FUNCTION_BLOCK "FB_Chute2PEC"
{ S7_Optimized_Access := 'TRUE' }
VERSION : 0.1
// ATTRIBUTES
// AUTO_NUMBER = True
// BLOCK_NUMBER = 204
// END_ATTRIBUTES
   VAR_INPUT
      iUDT_ChuteConfiguration { ExternalAccessible := 'False'; ExternalVisible := 'False'; ExternalWritable := 'False'} : "UDT_Chute2PECConfiguration";   // Chute Configuration structure
      iUDT_UpstreamConveyorStatus { ExternalAccessible := 'False'; ExternalVisible := 'False'; ExternalWritable := 'False'} : "UDT_CommonStatus";   // Upstream conveyor status
      ix_PECFull { ExternalAccessible := 'False'; ExternalVisible := 'False'; ExternalWritable := 'False'} : Bool;   // TRUE when Chute Full photoeye is not blocked
      ix_PECHalfFull { ExternalAccessible := 'False'; ExternalVisible := 'False'; ExternalWritable := 'False'} : Bool;   // TRUE when Chute Half Full photoeye is not blocked
      ix_Disabled { ExternalAccessible := 'False'; ExternalVisible := 'False'; ExternalWritable := 'False'} : Bool;   // TRUE when chute is disabled
      ix_HardwareOk { ExternalAccessible := 'False'; ExternalVisible := 'False'; ExternalWritable := 'False'} : Bool;   // TRUE when chute hardware is Ok
      iudi_DelayHardwareOK { ExternalAccessible := 'False'; ExternalVisible := 'False'; ExternalWritable := 'False'} : UDInt;   // Time to delay for hardware ok signal
   END_VAR

   VAR_OUTPUT
      qx_Lamp { ExternalAccessible := 'False'; ExternalVisible := 'False'; ExternalWritable := 'False'} : Bool;   // Output Chute Lamp half full/ full
      qUDT_HMIStatus { ExternalAccessible := 'False'; ExternalVisible := 'False'; ExternalWritable := 'False'} : "UDT_Chute2PECStatus";   // HMI status structure
      qUDT_Status { ExternalAccessible := 'False'; ExternalVisible := 'False'; ExternalWritable := 'False'} : "UDT_CommonStatus";   // Common status structure
   END_VAR

   VAR_IN_OUT
      iqUDT_EquipmentControl : "UDT_EquipmentControl";   // Equipment control structure
      iqUDT_UpstreamConveyorHandshake : "UDT_ConveyorHandshake";   // Upstream handshake structure
      iqUDT_Statistics : "UDT_Chute2PECStatistics";   // Statistics structure
   END_VAR

   VAR
      sUDT_HMIStatus { ExternalAccessible := 'False'; ExternalVisible := 'False'; ExternalWritable := 'False'; S7_SetPoint := 'False'} : "UDT_Chute2PECStatus";   // HMI status structure
      sUDT_CommonStatus { ExternalAccessible := 'False'; ExternalVisible := 'False'; ExternalWritable := 'False'; S7_SetPoint := 'False'} : "UDT_CommonStatus";   // Common status structure
      sUDT_CommonStatusOld { ExternalAccessible := 'False'; ExternalVisible := 'False'; ExternalWritable := 'False'; S7_SetPoint := 'False'} : "UDT_CommonStatus";   // Auxiliary status structure
      sFB_HardwareOk { ExternalAccessible := 'False'; ExternalVisible := 'False'; ExternalWritable := 'False'; S7_SetPoint := 'False'} : "FB_TimerOnOffDelay";   // Timer on/off delay for hardware ok signal
      sFB_ChuteHalfFullDetectionDelay { ExternalAccessible := 'False'; ExternalVisible := 'False'; ExternalWritable := 'False'; S7_SetPoint := 'False'} : "FB_TimerOnOffDelay";   // Timer on/off delay for chute half  full detection
      sFB_ChuteFullDetectionDelay { ExternalAccessible := 'False'; ExternalVisible := 'False'; ExternalWritable := 'False'; S7_SetPoint := 'False'} : "FB_TimerOnOffDelay";   // Timer on/off delay for chute full detection
      sR_TRIG_HalfFull {InstructionName := 'R_TRIG'; LibVersion := '1.0'; ExternalAccessible := 'False'; ExternalVisible := 'False'; ExternalWritable := 'False'; S7_SetPoint := 'False'} : R_TRIG;   // Rising edge trigger on chute half full signal
      sR_TRIG_Disabled {InstructionName := 'R_TRIG'; LibVersion := '1.0'; ExternalAccessible := 'False'; ExternalVisible := 'False'; ExternalWritable := 'False'; S7_SetPoint := 'False'} : R_TRIG;   // Rising edge trigger on chute disabled signal
      sR_TRIG_ChuteFull {InstructionName := 'R_TRIG'; LibVersion := '1.0'; ExternalAccessible := 'False'; ExternalVisible := 'False'; ExternalWritable := 'False'; S7_SetPoint := 'False'} : R_TRIG;   // Rising edge trigger on chute full signal
      sF_TRIG_UpdateStatus {InstructionName := 'F_TRIG'; LibVersion := '1.0'; ExternalAccessible := 'False'; ExternalVisible := 'False'; ExternalWritable := 'False'; S7_SetPoint := 'False'} : F_TRIG;   // Falling edge trigger on status change
      sx_Full { ExternalAccessible := 'False'; ExternalVisible := 'False'; ExternalWritable := 'False'} : Bool;   // Full status
      sx_HalfFull { ExternalAccessible := 'False'; ExternalVisible := 'False'; ExternalWritable := 'False'} : Bool;   // Half full status
   END_VAR


BEGIN
	(*
	----------------------------------------------------------------------------------------

	Version history:
	Date        | Version   | Author        | Remark
	----------------------------------------------------------------------------------------
	19/10/2021  | 0.1       | J. Krawczuk   | first release TIA 16.0
	29/10/2021  | 0.1       | M. Piela      | Design change, comments corrections
	14/01/2022  | 0.2       | G. Vlooswijk  | Fixed statistics reset
	30/07/2022  | 0.3       | G. Vlooswijk  | Removed running and energy save status for FedEx Scada
	21/02/2023  | 4.0       | F.Baten       | 4.0 Release TIA 17.5
	 *)

	REGION 1 - Timers

	    // Chute full detection timer
	    #sFB_ChuteFullDetectionDelay(iudi_OnDelayTime := #iUDT_ChuteConfiguration.FullDetectionTime,
	                                 iudi_OffDelayTime := #iUDT_ChuteConfiguration.FullReleaseTime,
	                                 ix_SignalToDelay := NOT #ix_PECFull,
	                                 qx_DelayedSignal => #sx_Full);

	    // Chute half full detection timer
	    #sFB_ChuteHalfFullDetectionDelay(iudi_OnDelayTime := #iUDT_ChuteConfiguration.HalfFullDetectionTime,
	                                     iudi_OffDelayTime := #iUDT_ChuteConfiguration.HalfFullReleaseTime,
	                                     ix_SignalToDelay := NOT #ix_PECHalfFull,
	                                     qx_DelayedSignal => #sx_HalfFull);

	    // Hardware ok signal delay
	    #sFB_HardwareOk(iudi_OnDelayTime := #iudi_DelayHardwareOK,
	                    ix_SignalToDelay := #ix_HardwareOk);


	END_REGION

	REGION 2 - Stop upstream conveyor

	    // Stop upstream conveyor when chute is full or disabled
	    #iqUDT_UpstreamConveyorHandshake.RTR := NOT #sx_Full AND NOT #ix_Disabled AND #sFB_HardwareOk.qx_DelayedSignal;

	END_REGION

	REGION 3 - Update output

	    // Update the outputs
	    #qx_Lamp := #sx_Full OR (#sx_HalfFull AND "DB_Memory".Clock_1Hz);

	END_REGION

	REGION 4 - Status

	    // Update chute full specific status
	    #sUDT_HMIStatus.Specific.ChuteFull := #sx_Full AND #sFB_HardwareOk.qx_DelayedSignal;

	    // Update chute half full specific status
	    #sUDT_HMIStatus.Specific.ChuteHalfFull := #sx_HalfFull AND #sFB_HardwareOk.qx_DelayedSignal;

	    //Update chute disabled specific status
	    #sUDT_HMIStatus.Specific.ChuteDisabled := #ix_Disabled AND #sFB_HardwareOk.qx_DelayedSignal;

	    // Update common safety stop
	    #sUDT_CommonStatus.SafetyStop := #iUDT_UpstreamConveyorStatus.SafetyStop;

	    // Update common automatic on
	    #sUDT_CommonStatus.AutoON := #iUDT_UpstreamConveyorStatus.AutoON;

	    // Update common stopped
	    #sUDT_CommonStatus.Stopped := #iUDT_UpstreamConveyorStatus.Stopped;

	    // Update HMI status number for chute disabled
	    IF #sUDT_HMIStatus.Specific.ChuteDisabled AND NOT #sUDT_CommonStatus.SafetyStop
	    THEN
	        #sUDT_HMIStatus.Status := "DB_HMIStatusConfiguration".DisableByManagement;

	    END_IF;

	    // Update HMI status number for chute half full
	    IF #sUDT_HMIStatus.Specific.ChuteHalfFull AND NOT #sUDT_CommonStatus.SafetyStop
	    THEN
	        #sUDT_HMIStatus.Status := "DB_HMIStatusConfiguration".ChuteHalfFull;

	    END_IF;

	    // Update HMI status number for chute full
	    IF #sUDT_HMIStatus.Specific.ChuteFull AND NOT #sUDT_CommonStatus.SafetyStop
	    THEN
	        #sUDT_HMIStatus.Status := "DB_HMIStatusConfiguration".ChuteFull;

	    END_IF;

	    // Collecting F_TRIG on chute full, chute half full or chute disabled status to update common status
	    #sF_TRIG_UpdateStatus(CLK := #sUDT_HMIStatus.Specific.ChuteFull
	                          OR #sUDT_HMIStatus.Specific.ChuteDisabled
	                          OR #sUDT_HMIStatus.Specific.ChuteHalfFull);

	    // HMI status number calculation
	    IF #sUDT_CommonStatusOld <> #sUDT_CommonStatus OR #sF_TRIG_UpdateStatus.Q
	    THEN

	        // Update auto on status number
	        IF #sUDT_CommonStatus.AutoON
	        THEN
	            #sUDT_HMIStatus.Status := "DB_HMIStatusConfiguration".AutoON;

	        END_IF;

	        IF #sUDT_CommonStatus.Stopped
	        THEN
	            #sUDT_HMIStatus.Status := "DB_HMIStatusConfiguration".Stopped;

	        END_IF;

	        IF #sUDT_CommonStatus.SafetyStop
	        THEN
	            #sUDT_HMIStatus.Status := "DB_HMIStatusConfiguration".SafetyStop;

	        END_IF;

	        // Copy common status structure to the old common status structure
	        #sUDT_CommonStatusOld := #sUDT_CommonStatus;
	        #qUDT_Status := #sUDT_CommonStatus;

	    END_IF;

	    #qUDT_HMIStatus := #sUDT_HMIStatus;

	END_REGION

	REGION 5 - Statistics

	    // Chute full R_TRIG for statistics purpose
	    #sR_TRIG_ChuteFull(CLK := #sUDT_HMIStatus.Specific.ChuteFull);

	    // Chute full statistics
	    IF #sUDT_HMIStatus.Specific.ChuteFull
	        OR #iqUDT_EquipmentControl.Command.ResetData
	    THEN
	        "FC_Statistics"(ix_Reset := #iqUDT_EquipmentControl.Command.ResetData,
	                        ix_Activate := #sUDT_HMIStatus.Specific.ChuteFull,
	                        ix_RTrigActivate := #sR_TRIG_ChuteFull.Q,
	                        iqUDT_Statistics := #iqUDT_Statistics.ChuteFull);

	    END_IF;

	    // Chute disabled R_TRIG for statistics purpose
	    #sR_TRIG_Disabled(CLK := #sUDT_HMIStatus.Specific.ChuteDisabled);

	    // Chute disabled statistics
	    IF #sUDT_HMIStatus.Specific.ChuteDisabled
	        OR #iqUDT_EquipmentControl.Command.ResetData
	    THEN
	        "FC_Statistics"(ix_Reset := #iqUDT_EquipmentControl.Command.ResetData,
	                        ix_Activate := #sUDT_HMIStatus.Specific.ChuteDisabled,
	                        ix_RTrigActivate := #sR_TRIG_Disabled.Q,
	                        iqUDT_Statistics := #iqUDT_Statistics.ChuteDisabled);

	    END_IF;

	    // Chute half full R_TRIG for statistics purpose
	    #sR_TRIG_HalfFull(CLK := #sUDT_HMIStatus.Specific.ChuteHalfFull);

	    // Chute half full statistics
	    IF #sUDT_HMIStatus.Specific.ChuteHalfFull
	        OR #iqUDT_EquipmentControl.Command.ResetData
	    THEN

	        "FC_Statistics"(ix_Reset := #iqUDT_EquipmentControl.Command.ResetData,
	                        ix_Activate := #sUDT_HMIStatus.Specific.ChuteHalfFull,
	                        ix_RTrigActivate := #sR_TRIG_HalfFull.Q,
	                        iqUDT_Statistics := #iqUDT_Statistics.ChuteHalfFull);

	    END_IF;

	END_REGION

	REGION 6 - Equipment Report

	    "FC_EquipmentReport"(iUDT_Status := #sUDT_CommonStatus,
	                         iqUDT_Control := #iqUDT_EquipmentControl);

	END_REGION
END_FUNCTION_BLOCK

FUNCTION_BLOCK "FB_PendantVT100"
{ S7_Optimized_Access := 'TRUE' }
VERSION : 0.1
// ATTRIBUTES
// AUTO_NUMBER = True
// BLOCK_NUMBER = 222
// END_ATTRIBUTES
   VAR_INPUT
      iUDT_Configuration { ExternalAccessible := 'False'; ExternalVisible := 'False'; ExternalWritable := 'False'} : "UDT_PendantVT100Configuration" := ([16#001B, 16#005B, 16#0031, 16#003B, 16#0033, 16#0048, 16#006D, 16#0000], [16#001B, 16#005B, 16#0032, 16#003B, 16#0035, 16#0048, 16#006D, 16#0000], (), (), ());
      iUDT_PendantInputs { ExternalAccessible := 'False'; ExternalVisible := 'False'; ExternalWritable := 'False'} : "UDT_PendantVT100InBytes";   //   Input Bytes 1,2 and 3 of HW Config
      ix_HMIDivertSelectionEnabled { ExternalAccessible := 'False'; ExternalVisible := 'False'; ExternalWritable := 'False'} : Bool;   //   When 'TRUE' The divert selection screen is activated from the HMI
      ix_SimulationModeActive { ExternalAccessible := 'False'; ExternalVisible := 'False'; ExternalWritable := 'False'} : Bool;   //   When 'TRUE' Simulation mode active
      ix_LCDDS1 { ExternalAccessible := 'False'; ExternalVisible := 'False'; ExternalWritable := 'False'} : Bool;   //   When 'TRUE' Display is busy writing a message row 1
      ix_PowerOk { ExternalAccessible := 'False'; ExternalVisible := 'False'; ExternalWritable := 'False'} : Bool;   //   When 'TRUE' 24VDC available
      ix_ServiceMode { ExternalAccessible := 'False'; ExternalVisible := 'False'; ExternalWritable := 'False'} : Bool;   //   When 'TRUE' Service Mode ON
      ix_VFDRunFeedback { ExternalAccessible := 'False'; ExternalVisible := 'False'; ExternalWritable := 'False'} : Bool;   //   When 'TRUE' VFD Run
      ix_SorterSTOActive { ExternalAccessible := 'False'; ExternalVisible := 'False'; ExternalWritable := 'False'} : Bool;   //   VFD STO active feedback
      ix_SorterSS1Active { ExternalAccessible := 'False'; ExternalVisible := 'False'; ExternalWritable := 'False'} : Bool;   //   VFD SS1 active feedback
   END_VAR

   VAR_OUTPUT
      qUDT_Display { ExternalAccessible := 'False'; ExternalVisible := 'False'; ExternalWritable := 'False'} : "UDT_PendantVT100LCDOutBytes";   //   Display bytes
      qUDT_HMIStatus { ExternalAccessible := 'False'; ExternalVisible := 'False'; ExternalWritable := 'False'} : "UDT_PendantVT100Status";   //   Configuation variables for VT100 Radio Pendant
      qUDT_Status { ExternalAccessible := 'False'; ExternalVisible := 'False'; ExternalWritable := 'False'} : "UDT_CommonStatus";   //   Common status structure
   END_VAR

   VAR_IN_OUT
      iqUDT_EquipmentControl : "UDT_EquipmentControl";
      iqUDT_PendantInterface : "UDT_PendantVT100Interface";   //   Interface structure
      iqUDT_Statistics : "UDT_PendantVT100Statistics";   //   Staristic structure
      iq_ConveyorInterface : "UDT_ConveyorInterface";
   END_VAR

   VAR
      sUDT_Display { ExternalAccessible := 'False'; ExternalVisible := 'False'; ExternalWritable := 'False'; S7_SetPoint := 'False'} : "UDT_PendantVT100LCDOutBytes";   //    Array of 8 bytes for the display message
      sUDT_CommonStatus { ExternalAccessible := 'False'; ExternalVisible := 'False'; ExternalWritable := 'False'; S7_SetPoint := 'False'} : "UDT_CommonStatus";   //    Common status structure
      sUDT_CommonStatusOld { ExternalAccessible := 'False'; ExternalVisible := 'False'; ExternalWritable := 'False'; S7_SetPoint := 'False'} : "UDT_CommonStatus";   //    Common status structure
      sUDT_HMIStatus { ExternalAccessible := 'False'; ExternalVisible := 'False'; ExternalWritable := 'False'; S7_SetPoint := 'False'} : "UDT_PendantVT100Status";
      sUDT_PNDevice { ExternalAccessible := 'False'; ExternalVisible := 'False'; ExternalWritable := 'False'; S7_SetPoint := 'False'} : "UDT_PNDevice";   //    PN device info structure
      sFB_TimerOnOffDelayCheckSupply { ExternalAccessible := 'False'; ExternalVisible := 'False'; ExternalWritable := 'False'; S7_SetPoint := 'False'} : "FB_TimerOnOffDelay";
      sF_TRIG_Servicemode {InstructionName := 'F_TRIG'; LibVersion := '1.0'; ExternalAccessible := 'False'; ExternalVisible := 'False'; ExternalWritable := 'False'; S7_SetPoint := 'False'} : F_TRIG;   //   Falling edge trigger service mode
      sF_TRIG_DisplayReady {InstructionName := 'F_TRIG'; LibVersion := '1.0'; ExternalAccessible := 'False'; ExternalVisible := 'False'; ExternalWritable := 'False'; S7_SetPoint := 'False'} : F_TRIG;   //   Falling edge trigger display ready
      sR_TRIG_RunCommand {InstructionName := 'R_TRIG'; LibVersion := '1.0'; ExternalAccessible := 'False'; ExternalVisible := 'False'; ExternalWritable := 'False'; S7_SetPoint := 'False'} : R_TRIG;   //   Rising edge trigger run command
      sR_TRIG_PNReceiverNotOnline {InstructionName := 'R_TRIG'; LibVersion := '1.0'; ExternalAccessible := 'False'; ExternalVisible := 'False'; ExternalWritable := 'False'; S7_SetPoint := 'False'} : R_TRIG;   //   Rising edge trigger PN receiver not online
      sR_TRIG_PNReceiverError {InstructionName := 'R_TRIG'; LibVersion := '1.0'; ExternalAccessible := 'False'; ExternalVisible := 'False'; ExternalWritable := 'False'; S7_SetPoint := 'False'} : R_TRIG;   //   Rising edge trigger PN device error
      sR_TRIG_ControlHealthy {InstructionName := 'R_TRIG'; LibVersion := '1.0'; ExternalAccessible := 'False'; ExternalVisible := 'False'; ExternalWritable := 'False'; S7_SetPoint := 'False'} : R_TRIG;   //   Rising edge trigger control healthy
      sa_Int { ExternalAccessible := 'False'; ExternalVisible := 'False'; ExternalWritable := 'False'} : Struct   //   Integer structure
         Step { ExternalAccessible := 'False'; ExternalVisible := 'False'; ExternalWritable := 'False'; S7_SetPoint := 'True'} : Int;   //    Step of the message sequence
      END_STRUCT;
      sa_Bool { ExternalAccessible := 'False'; ExternalVisible := 'False'; ExternalWritable := 'False'} : Struct   //   Bool structure
         DivertUp { ExternalAccessible := 'False'; ExternalVisible := 'False'; ExternalWritable := 'False'} : Bool;   //    When 'TRUE' Any divert is up
         HardwareAvailable { ExternalAccessible := 'False'; ExternalVisible := 'False'; ExternalWritable := 'False'} : Bool;   //    When 'TRUE' Hardware available and ready to use
         PermissionRequested { ExternalAccessible := 'False'; ExternalVisible := 'False'; ExternalWritable := 'False'} : Bool;   //    When 'TRUE' Permission requested for horn to sound
         PermissionGranted { ExternalAccessible := 'False'; ExternalVisible := 'False'; ExternalWritable := 'False'} : Bool;   //    When 'TRUE' Horn sounded before start of VFD
         PowerOk { ExternalAccessible := 'False'; ExternalVisible := 'False'; ExternalWritable := 'False'} : Bool;   //    When 'TRUE' Power is present at receiver
         PNDeviceHealthy { ExternalAccessible := 'False'; ExternalVisible := 'False'; ExternalWritable := 'False'} : Bool;   //    When 'TRUE' Receiver is healthy
         RadioConnection { ExternalAccessible := 'False'; ExternalVisible := 'False'; ExternalWritable := 'False'} : Bool;   //    When 'TRUE' Initial connection with radio
         RunRequest { ExternalAccessible := 'False'; ExternalVisible := 'False'; ExternalWritable := 'False'} : Bool;   //    When 'TRUE' Request to run
         ServiceModeEngaged { ExternalAccessible := 'False'; ExternalVisible := 'False'; ExternalWritable := 'False'} : Bool;   //    True = Service mode is engaged
      END_STRUCT;
   END_VAR

   VAR_TEMP
      ti_index : Int;   //   temporary integer for loops
   END_VAR

   VAR CONSTANT
      cudi_PowerSupplyDelayTime : UDInt := 7000;   //   Power supply delay time [ms]
   END_VAR


BEGIN

	(*
	----------------------------------------------------------------------------------------

	Version history:
	Date        | Version   | Author        | Remark
	----------------------------------------------------------------------------------------
	14/04/2019  | 1.0       | S. Theocharis | first release TIA15.1
	11/09/2019  | 1.1       | S. Theocharis | update for UPS EMA Baseline
	04/11/2019  | 1.2       | S. Theocharis | Key Switch wired@safety input
	30/01/2020  | 3.0       | S. Theocharis | Different button for fast speed,
	                                        | code to activate diverters
	                                        | Status, statistics and equipement control
	                                        | structures added
	04/03/2020  | 3.1       | M. Piela      | Changed comments and subregions names, added constants to timers
	25/06/2020  | 3.2       | L. Klar       | Horn delay deleted
	07/07/2020  | 3.3       | M. Piela      | Delete unused signal from the interface, change condition to enable step 1
	                                        | in service mode
	07/07/2020  | 3.4       | M. Piela      | Added conditions to set the signaling request signal
	28/07/2020  | 3.5       | S. Theocharis | Changed input name
	11/08/2020  | 3.6       | S. Theocharis | Update the divert functionality
	03/06/2021  | 3.7       | S. Theocharis | Force to slow speed for missing pin at service point
	21/02/2023  | 4.0       | F.Baten       | 4.0 Release TIA 17.5
	*)

	REGION Notes
	(*

	Note1:
	 ib_Buttons.xxxxxx1 is  the signal when the associate button is pressed half way
	 ib_buttons.xxxxxx2 is  the signal when the associate button is pressed full

	 Not Pressed:                 Halfway Pressed                    Full way Pressed
	                             ib_Buttons.xxxxxx1 = TRUE           ib_Buttons.xxxxxx1 = TRUE
	                             ib_Buttons.xxxxxx2 = FALSE          ib_Buttons.xxxxxx2 = TRUE
	     ________
	     |      |                        ________
	     |      |                        |      |                       ________
	     |      |                        |      |                       |      |
	 ____|      |____                 ___|      |____                ___|      |____


	 Note2:
	 The block is designed for the following remote controller:
	 Danfoss TM70/1.13DC  (Ikusi)
	 https://www.danfoss.com/en/products/electronic-controls/dps/plus1-remote-controls/transmitters/legacy-handheld-transmitters/
	  *)
	END_REGION

	REGION 1 -  Get Receiver Profinet number

	    "FC_GetDevicePN"(is_PNDeviceName := #iUDT_Configuration.PNDeviceName,
	                     ix_SimulationModeActive := #ix_SimulationModeActive,
	                     iqUDT_PND := #sUDT_PNDevice);

	END_REGION

	REGION 2 - Reset errors

	    IF #iqUDT_EquipmentControl.Command.Reset                         // Reser errors when Reset from HMI or MCP is given
	    THEN
	        #sUDT_HMIStatus.Specific.PNSlaveNotOnline := FALSE;
	        #sUDT_HMIStatus.Specific.PNSlaveError := FALSE;
	        #sUDT_HMIStatus.Specific.CommunicationError := FALSE;          // Not in use
	    END_IF;

	END_REGION

	REGION 3 - Hardware checks
	    // PN Receiver will only be available after the delay, so the device has time for the initialisation
	    #sFB_TimerOnOffDelayCheckSupply(iudi_OnDelayTime := #cudi_PowerSupplyDelayTime,
	                                    ix_SignalToDelay := #ix_PowerOk,
	                                    ix_Enable := TRUE,
	                                    qx_DelayedSignal => #sa_Bool.PowerOk);

	    // Check if PN receiver device is online
	    IF NOT "DB_ProfinetDiagnostic".ProfinetNetworks[#sUDT_PNDevice.PNNetworknumber].DeviceStatus[#sUDT_PNDevice.PNDeviceNumber].DeviceState.Exist
	        AND NOT #ix_SimulationModeActive
	        AND #sa_Bool.PowerOk
	    THEN
	        #sUDT_HMIStatus.Specific.PNSlaveNotOnline := TRUE;
	    END_IF;

	    // Check if PN Receiver device has an error
	    IF "DB_ProfinetDiagnostic".ProfinetNetworks[#sUDT_PNDevice.PNNetworknumber].DeviceStatus[#sUDT_PNDevice.PNDeviceNumber].DeviceState.Error
	        AND NOT #ix_SimulationModeActive
	        AND #sa_Bool.PowerOk
	    THEN
	        #sUDT_HMIStatus.Specific.PNSlaveError := TRUE;
	    END_IF;

	    // Set bit when PN Receiver device is healthy (online and no error)
	    #sa_Bool.PNDeviceHealthy := NOT #sUDT_HMIStatus.Specific.PNSlaveNotOnline
	    AND NOT #sUDT_HMIStatus.Specific.PNSlaveError
	    AND #sUDT_PNDevice.PNDeviceFound
	    AND #sa_Bool.PowerOk;

	    // Set hardware available bit when all conditions are met
	    #sa_Bool.HardwareAvailable := (#sa_Bool.PowerOk
	    AND #sa_Bool.PNDeviceHealthy)
	    OR #ix_SimulationModeActive;

	END_REGION

	REGION 4 -  Detect service mode selection changes

	    //static memory to engage the service mode. Only when the sorter is standstill
	    IF #sa_Bool.HardwareAvailable AND #ix_ServiceMode AND NOT #ix_VFDRunFeedback
	    THEN
	        #sa_Bool.ServiceModeEngaged := TRUE;
	    END_IF;

	    //disengage service mode when hardware is not available or switch is off
	    IF NOT #sa_Bool.HardwareAvailable OR NOT #ix_ServiceMode
	    THEN
	        #sa_Bool.ServiceModeEngaged := FALSE;
	    END_IF;

	    //service mode to interface
	    #iqUDT_PendantInterface.ServiceModeEngaged := #sa_Bool.ServiceModeEngaged;


	    //Detect falling edge of service mode
	    #sF_TRIG_Servicemode(CLK := #sa_Bool.ServiceModeEngaged);

	END_REGION

	REGION 5 -  Service mode

	    IF #sa_Bool.ServiceModeEngaged
	    THEN

	        REGION 5.1 - Detect Tx connection & LCD readiness to receive message

	            #sR_TRIG_ControlHealthy(CLK := #iUDT_PendantInputs.Stop_NC);//Rising edge of communication

	            //set radio Tx-Rx connection
	            IF #sR_TRIG_ControlHealthy.Q
	            THEN    (* or replace it directly with the input #iudt_PendantInputs.Stop_NO) *)
	                #sa_Bool.RadioConnection := True;
	            END_IF;

	            #sF_TRIG_DisplayReady(CLK := #ix_LCDDS1);//LCD Status Signal. When ix_LCD_DS1 is False, the LCD is ready to receive a new message

	        END_REGION

	        REGION 5.2 - LCD messages
	            //First communication established. Activate message one to move cursor in the begin of line 1

	            IF #sa_Bool.RadioConnection
	            THEN
	                #sa_Int.Step := 1;           // step 1 - new message is activated
	                #sa_Bool.RadioConnection := FALSE;
	            END_IF;

	            //reset variables for display. that can be used to move the step to eg 98 and there reset the variables and move the step to 0 again
	            IF NOT #iUDT_PendantInputs.Stop_NC
	            THEN
	                // #st_Int.Step := 98;
	                FOR #ti_index := 0 TO 7 BY 1 DO
	                    #qUDT_Display."Byte"[#ti_index] := b#16#0;
	                    #sUDT_Display."Byte"[#ti_index] := b#16#0;
	                END_FOR;
	            END_IF;

	            // Screen  Messages
	            CASE #sa_Int.Step OF

	                1: // Move Cursor in the Start Point
	                    #sUDT_Display."Byte" := #iUDT_Configuration.Line1Cursor;  // message
	                    #sa_Int.Step := 2;                                 //  is written static memory

	                2: // when display is not busy write the output
	                    IF NOT #ix_LCDDS1
	                    THEN
	                        #qUDT_Display."Byte" := #sUDT_Display."Byte";
	                        #sa_Int.Step := 3;    // move to next step
	                    END_IF;

	                3: //Write PLC name
	                    FOR #ti_index := 0 TO 7 BY 1 DO
	                        #sUDT_Display."Byte"[#ti_index] := CHAR_TO_BYTE(#iUDT_Configuration.DisplayName[#ti_index + 1]);
	                    END_FOR;
	                    #sa_Int.Step := 4;     //move to next step

	                4: //when display is not busy write the output
	                    IF #sF_TRIG_DisplayReady.Q
	                    THEN   (* may need to be replaced with :NOT #ix_LCD_DS1 *)
	                        #qUDT_Display."Byte" := #sUDT_Display."Byte";
	                        #sa_Int.Step := 99;// move to next step
	                    END_IF;
	            END_CASE;

	        END_REGION

	        REGION 5.3 - Output to the sorter control function
	            //Stop Button
	            #iqUDT_PendantInterface.PendantStopHealthy := #iUDT_PendantInputs.Stop_NC AND NOT #iUDT_PendantInputs.Stop_NO;

	            // Reset - Control On
	            #iqUDT_PendantInterface.PendantReset := #iUDT_PendantInputs.ResetButton1;

	        END_REGION

	        REGION 5.4 - Motion control
	            // STO request to safety program
	            #iqUDT_PendantInterface.RequestSTO := #iUDT_PendantInputs.PB_Speed1 OR #iUDT_PendantInputs.PB_Speed2;

	            //Run reuqest condition
	            #sa_Bool.RunRequest := (#iUDT_PendantInputs.PB_Speed2 XOR #iUDT_PendantInputs.PB_Speed1) AND NOT #sa_Bool.DivertUp;

	            //Check permission to run after horn sounded
	            IF #iUDT_Configuration.HornRequest
	            THEN

	                //Detect new run request
	                #sR_TRIG_RunCommand(CLK := #sa_Bool.RunRequest AND NOT #ix_VFDRunFeedback);

	                //On the positie edge of the new run command which requires permission set the control request and reset the permissiong granted bit
	                IF #sR_TRIG_RunCommand.Q AND NOT #ix_SorterSS1Active AND NOT #iq_ConveyorInterface.InternalErrorVFD
	                THEN
	                    #iqUDT_EquipmentControl.Request.SignalingRequest := TRUE;
	                    #sa_Bool.PermissionRequested := TRUE;
	                    #sa_Bool.PermissionGranted := FALSE;
	                END_IF;

	                //when the requested memory is true but the control request is false, it means that the horn sounded and the permission to run is granted again
	                IF #sa_Bool.PermissionRequested AND NOT #iqUDT_EquipmentControl.Request.SignalingRequest
	                THEN
	                    #sa_Bool.PermissionRequested := FALSE;
	                    #sa_Bool.PermissionGranted := TRUE;
	                END_IF;

	            ELSE  //when horn request is deactivated via the configuration
	                #sa_Bool.PermissionGranted := TRUE;
	                #sa_Bool.PermissionRequested := FALSE;
	            END_IF;

	            //assign commands to run and speed only when associate button is pressed and not divert is detected up
	            #iqUDT_PendantInterface.CmdRun := NOT #ix_SorterSTOActive AND #sa_Bool.PermissionGranted AND #sa_Bool.RunRequest;

	            #iqUDT_PendantInterface.LowSpeedSelected := (#iUDT_PendantInputs.PB_Speed1
	            OR
	            (#iUDT_PendantInputs.PB_Speed2 AND #iqUDT_PendantInterface.ForceLowSpeed))
	            AND #sa_Bool.PermissionGranted
	            AND #sa_Bool.RunRequest;


	            #iqUDT_PendantInterface.ManualSpeedSelected := (#iUDT_PendantInputs.PB_Speed2 AND NOT #iqUDT_PendantInterface.ForceLowSpeed)
	            AND #sa_Bool.PermissionGranted
	            AND #sa_Bool.RunRequest;

	        END_REGION

	    ELSE

	        REGION 5.7 - Reset interface bits when service mode is disengaged

	            #iqUDT_PendantInterface.CmdRun := FALSE;
	            #iqUDT_PendantInterface.LowSpeedSelected := FALSE;
	            #iqUDT_PendantInterface.ManualSpeedSelected := FALSE;
	            #iqUDT_PendantInterface.PendantReset := FALSE;
	            #iqUDT_PendantInterface.PendantStopHealthy := FALSE;


	        END_REGION

	    END_IF;

	END_REGION

	REGION 6 Divert functionality

	    #iqUDT_PendantInterface.CmdDivert := #iUDT_PendantInputs.PB_Divert
	    AND #sa_Bool.ServiceModeEngaged
	    AND #ix_HMIDivertSelectionEnabled
	    AND NOT #ix_VFDRunFeedback;

	END_REGION


	REGION 7 - Statistics

	    // Create trigger on error and create statistics for profinet slave not online
	    #sR_TRIG_PNReceiverNotOnline(CLK := #sUDT_HMIStatus.Specific.PNSlaveNotOnline);

	    IF #iqUDT_EquipmentControl.Command.ResetData OR #sUDT_HMIStatus.Specific.PNSlaveNotOnline
	    THEN

	        "FC_Statistics"(ix_Reset := #iqUDT_EquipmentControl.Command.ResetData,
	                        ix_Activate := #sUDT_HMIStatus.Specific.PNSlaveNotOnline,
	                        ix_RTrigActivate := #sR_TRIG_PNReceiverNotOnline.Q,
	                        iqUDT_Statistics := #iqUDT_Statistics.PNSlaveNotOnline);
	    END_IF;

	    // Create trigger on error and create statistics for profinet slave error
	    #sR_TRIG_PNReceiverError(CLK := #sUDT_HMIStatus.Specific.PNSlaveError);

	    IF #iqUDT_EquipmentControl.Command.ResetData OR #sUDT_HMIStatus.Specific.PNSlaveError
	    THEN

	        "FC_Statistics"(ix_Reset := #iqUDT_EquipmentControl.Command.ResetData,
	                        ix_Activate := #sUDT_HMIStatus.Specific.PNSlaveError,
	                        ix_RTrigActivate := #sR_TRIG_PNReceiverError.Q,
	                        iqUDT_Statistics := #iqUDT_Statistics.PNSlaveError);
	    END_IF;

	END_REGION

	REGION 8 - Status

	    //update status of service mode engaged
	    #sUDT_HMIStatus.Specific.ServiceModeEngaged := #sa_Bool.ServiceModeEngaged;

	    //prepare commont status for equipment report
	    #sUDT_CommonStatus.Error := (#sUDT_HMIStatus.Specific.PNSlaveError OR #sUDT_HMIStatus.Specific.PNSlaveNotOnline OR #sUDT_HMIStatus.Specific.CommunicationError);

	    // HMI status update
	    IF #sUDT_CommonStatusOld <> #sUDT_CommonStatus      // update on change
	    THEN
	        // HMI status initialization
	        #sUDT_HMIStatus.Status := 0;

	        // HMI status calculation
	        IF #sUDT_HMIStatus.Specific.PNSlaveError OR #sUDT_HMIStatus.Specific.PNSlaveNotOnline
	        THEN
	            #sUDT_HMIStatus.Status := "DB_HMIStatusConfiguration".ProfinetError;
	        END_IF;
	    END_IF;

	    #qUDT_HMIStatus := #sUDT_HMIStatus;                          // Copy HMI status to output
	    #sUDT_CommonStatusOld := #sUDT_CommonStatus;                 // Copy status to memory
	    #qUDT_Status := #sUDT_CommonStatus;                          // Copy status to output

	END_REGION

	REGION 9 - Report to control block
	    // Function to manage report between control block and conveyor block
	    "FC_EquipmentReport"(iUDT_Status := #sUDT_CommonStatus,
	                         iqUDT_Control := #iqUDT_EquipmentControl);

	END_REGION
END_FUNCTION_BLOCK

FUNCTION_BLOCK "FB_ConnectionCheck"
{ S7_Optimized_Access := 'TRUE' }
VERSION : 3.2
// ATTRIBUTES
// AUTO_NUMBER = True
// BLOCK_NUMBER = 205
// END_ATTRIBUTES
   VAR_INPUT
      ib_Watchdog { ExternalAccessible := 'False'; ExternalVisible := 'False'; ExternalWritable := 'False'} : Byte;   // Input watchdog
      ix_Trigger100ms { ExternalAccessible := 'False'; ExternalVisible := 'False'; ExternalWritable := 'False'} : Bool;   // Cycled 100 ms trigger
   END_VAR

   VAR_OUTPUT
      qb_Watchdog { ExternalAccessible := 'False'; ExternalVisible := 'False'; ExternalWritable := 'False'} : Byte;   // Generated watchdog
   END_VAR

   VAR_IN_OUT
      iqudt_ConnectionStatus : "UDT_ConnectStatus";   // Connection status
   END_VAR

   VAR
      s_FB_ConnectionFaultTimerOnDelay { ExternalAccessible := 'False'; ExternalVisible := 'False'; ExternalWritable := 'False'; S7_SetPoint := 'False'} : "FB_TimerOnOffDelay";   // Connection fault timer on delay
      sb_InWatchdogOld { ExternalAccessible := 'False'; ExternalVisible := 'False'; ExternalWritable := 'False'} : Byte;   // Watch dog old
      sb_GeneratedWatchdog { ExternalAccessible := 'False'; ExternalVisible := 'False'; ExternalWritable := 'False'} : Byte;   // Generated watchdog
      sx_SetConnectionFaultTimer { ExternalAccessible := 'False'; ExternalVisible := 'False'; ExternalWritable := 'False'} : Bool;   // Set connection fault timer
      sx_ConnectionFault { ExternalAccessible := 'False'; ExternalVisible := 'False'; ExternalWritable := 'False'} : Bool;   // Connection faulr
   END_VAR

   VAR CONSTANT
      cudi_ConnectionFaultOnDelay : UDInt := 10000;   // Connection On Delay
   END_VAR


BEGIN
	(*
	----------------------------------------------------------------------------------------
	|                                                                                      |
	|  Copyright  2023             FORTNA Europe BV                                        |
	|  All Rights Reserved         Netherlands                                             |
	|                                                                                      |
	----------------------------------------------------------------------------------------

	Version history:
	Date        | Version   | Author        | Remark
	----------------------------------------------------------------------------------------
	31/03/2022  | 3.0       | M. Piela      | First release TIA 16
	06/09/2023  | 3.1       | S. Nikodem    | Added watchdog generations on output
	11/09/2023  | 3.2       | S. Theocharis | Corrected variable prefixes
	*)

	REGION 1 - Connection check

	    #sx_SetConnectionFaultTimer := (#ib_Watchdog = #sb_InWatchdogOld);

	    IF #ib_Watchdog <> #sb_InWatchdogOld
	    THEN
	        #sb_InWatchdogOld := #ib_Watchdog;
	    END_IF;

	    #s_FB_ConnectionFaultTimerOnDelay(iudi_OnDelayTime := #cudi_ConnectionFaultOnDelay,
	                                      ix_SignalToDelay := #sx_SetConnectionFaultTimer,
	                                      ix_Enable := TRUE,
	                                      qx_DelayedSignal => #sx_ConnectionFault);

	END_REGION

	REGION 2 - Status update

	    #iqudt_ConnectionStatus.Specific.CommunicationFault := #sx_ConnectionFault;
	    #iqudt_ConnectionStatus.Specific.Connected := NOT #sx_ConnectionFault;

	    IF #sx_ConnectionFault
	    THEN
	        #iqudt_ConnectionStatus.Status := "DB_HMIStatusConfiguration".CommunicationError;
	    END_IF;

	    IF NOT #sx_ConnectionFault
	    THEN
	        #iqudt_ConnectionStatus.Status := "DB_HMIStatusConfiguration".AutoON;
	    END_IF;

	END_REGION

	REGION 3 - Watchdog generations

	    //Watchdog counter to be updated after every 100 msec
	    IF #ix_Trigger100ms THEN

	        IF #sb_GeneratedWatchdog >= 255 OR #sb_GeneratedWatchdog < 0
	        THEN
	            #sb_GeneratedWatchdog := 0;
	        END_IF;

	        #sb_GeneratedWatchdog := INT_TO_BYTE(BYTE_TO_INT(#sb_GeneratedWatchdog) + 1);

	    END_IF;

	    //Copy value
	    #qb_Watchdog := #sb_GeneratedWatchdog;

	END_REGION
END_FUNCTION_BLOCK

FUNCTION_BLOCK "FB_ControlPowerGroupWOR"
TITLE = Control Power Group
{ S7_Optimized_Access := 'TRUE' }
AUTHOR : CesarLeite
VERSION : 3.0
// ATTRIBUTES
// AUTO_NUMBER = True
// BLOCK_NUMBER = 206
// END_ATTRIBUTES
//This block is used to monitoring the 24V power supplies.
   VAR_INPUT
      ix_PowerSupplyOK { ExternalAccessible := 'False'; ExternalVisible := 'False'; ExternalWritable := 'False'} : Bool;   //   TRUE if power supply is OK
      ix_HardwareOK { ExternalAccessible := 'False'; ExternalVisible := 'False'; ExternalWritable := 'False'} : Bool;   //  Hardware is ok
      iudi_DelayPowerSupplyOK { ExternalAccessible := 'False'; ExternalVisible := 'False'; ExternalWritable := 'False'} : UDInt;   //  Time to delay power supply ok signal
   END_VAR

   VAR_OUTPUT
      qUDT_HMIStatus { ExternalAccessible := 'False'; ExternalVisible := 'False'; ExternalWritable := 'False'} : "UDT_ControlPowerGroupWORStatus";   //   HMI status structure
      qUDT_Status { ExternalAccessible := 'False'; ExternalVisible := 'False'; ExternalWritable := 'False'} : "UDT_CommonStatus";   //   Common status structure
      qx_ResetPowerSupply { ExternalAccessible := 'False'; ExternalVisible := 'False'; ExternalWritable := 'False'} : Bool;
   END_VAR

   VAR_IN_OUT
      iqUDT_EquipmentControl : "UDT_EquipmentControl";   //   CIP Equipment control
      iqUDT_Statistics : "UDT_ControlPowerGroupWORStatistics";   //   CPG Statistics structure
   END_VAR

   VAR
      sUDT_HMIStatus { ExternalAccessible := 'False'; ExternalVisible := 'False'; ExternalWritable := 'False'; S7_SetPoint := 'False'} : "UDT_ControlPowerGroupWORStatus";   //   HMI status structure
      sUDT_CommonStatus { ExternalAccessible := 'False'; ExternalVisible := 'False'; ExternalWritable := 'False'; S7_SetPoint := 'False'} : "UDT_CommonStatus";   //   Common status structure
      sUDT_CommonStatusOld { ExternalAccessible := 'False'; ExternalVisible := 'False'; ExternalWritable := 'False'; S7_SetPoint := 'False'} : "UDT_CommonStatus";   //   Auxiliary status structure
      sFB_DelayInput { ExternalAccessible := 'False'; ExternalVisible := 'False'; ExternalWritable := 'False'; S7_SetPoint := 'False'} : "FB_TimerOnOffDelay";
      sFB_DelayHardwarOK { ExternalAccessible := 'False'; ExternalVisible := 'False'; ExternalWritable := 'False'; S7_SetPoint := 'False'} : "FB_TimerOnOffDelay";
      sFB_DelayResetPowerSupply { ExternalAccessible := 'False'; ExternalVisible := 'False'; ExternalWritable := 'False'; S7_SetPoint := 'False'} : "FB_TimerOnOffDelay";
      sR_TRIG_Error {InstructionName := 'R_TRIG'; LibVersion := '1.0'; ExternalAccessible := 'False'; ExternalVisible := 'False'; ExternalWritable := 'False'; S7_SetPoint := 'False'} : R_TRIG;   //   Rising edge for error
      sx_ResetPowerSupply { ExternalAccessible := 'False'; ExternalVisible := 'False'; ExternalWritable := 'False'} : Bool;
   END_VAR

   VAR CONSTANT
      cudi_ResetPowerSupplyTime : UDInt := 3000;
   END_VAR


BEGIN
	(*
	----------------------------------------------------------------------------------------

	Version history:
	Date        | Version   | Author        | Remark
	----------------------------------------------------------------------------------------
	12/10/2021  | 0.1       | J.Krawczuk    | first release TIA 15.1
	12/11/2021  | 0.2       | S.Theocharis  | Change code to match names of new status UDT
	06/06/2021  | 0.3       | K. Pokorski   | Added PSC reset output
	25/07/2022  | 0.4       | M.Piela       | Change running status to AutoOn
	21/02/2023  | 4.0       | F.Baten       | 4.0 Release TIA 17.5
	*)

	REGION 1 - Power Supply monitoring

	    // Delay on power supply ok signal to mask wrong SPG power errors
	    #sFB_DelayInput(iudi_OnDelayTime := 0,
	                    iudi_OffDelayTime := #iudi_DelayPowerSupplyOK,
	                    ix_SignalToDelay := #ix_PowerSupplyOK);

	    #sFB_DelayHardwarOK(iudi_OnDelayTime := #iudi_DelayPowerSupplyOK,
	                        iudi_OffDelayTime := 0,
	                        ix_SignalToDelay := #ix_HardwareOK);

	END_REGION

	REGION 2 - Reset

	    #sx_ResetPowerSupply := FALSE;
	    IF #iqUDT_EquipmentControl.Command.Reset
	    THEN
	        #sUDT_HMIStatus.Specific.PowerSuppliesError := FALSE;
	        #sx_ResetPowerSupply := TRUE;
	    END_IF;

	    #sFB_DelayResetPowerSupply(iudi_OffDelayTime := #cudi_ResetPowerSupplyTime,
	                               ix_SignalToDelay := #sx_ResetPowerSupply,
	                               qx_DelayedSignal => #qx_ResetPowerSupply);


	END_REGION

	REGION 3 - Status

	    // Set error state if there is an error with the power supply
	    IF NOT #sFB_DelayInput.qx_DelayedSignal            // Delayed power ok signal
	        AND #sFB_DelayHardwarOK.qx_DelayedSignal       // Delayed hardware ok signal
	    THEN
	        #sUDT_HMIStatus.Specific.PowerSuppliesError := TRUE;

	    END_IF;

	    // R_TRIG for statistics purposes
	    #sR_TRIG_Error(CLK := #sUDT_HMIStatus.Specific.PowerSuppliesError);

	END_REGION

	REGION 4 - Statistics

	    //  Error statistics
	    IF #sUDT_HMIStatus.Specific.PowerSuppliesError
	        OR #iqUDT_EquipmentControl.Command.ResetData
	    THEN

	        "FC_Statistics"(ix_Reset := #iqUDT_EquipmentControl.Command.ResetData,
	                        ix_Activate := #sUDT_HMIStatus.Specific.PowerSuppliesError,
	                        ix_RTrigActivate := #sR_TRIG_Error.Q,
	                        iqUDT_Statistics := #iqUDT_Statistics.PowerSupplyError);

	    END_IF;

	END_REGION

	REGION 5 - Status Update

	    #sUDT_CommonStatus.Error := #sUDT_HMIStatus.Specific.PowerSuppliesError;
	    #sUDT_CommonStatus.AutoON := NOT #sUDT_HMIStatus.Specific.PowerSuppliesError;


	    // HMI status update
	    IF #sUDT_CommonStatusOld <> #sUDT_CommonStatus                    // update on change
	    THEN

	        // HMI status initialization
	        #sUDT_HMIStatus.Status := 0;

	        IF #sUDT_CommonStatus.AutoON
	        THEN
	            #sUDT_HMIStatus.Status := "DB_HMIStatusConfiguration".AutoON;
	        END_IF;


	        IF #sUDT_CommonStatus.Error                                    // Error
	        THEN

	            #sUDT_HMIStatus.Status := "DB_HMIStatusConfiguration".Error;

	        END_IF;


	        #qUDT_Status := #sUDT_CommonStatus;                           // Copy status to output
	        #sUDT_CommonStatusOld := #sUDT_CommonStatus;                  // Copy status to memory

	    END_IF;
	    #qUDT_HMIStatus := #sUDT_HMIStatus;                               // Copy HMI status to output


	END_REGION

	REGION 6 - Report to control block

	    // Function to manage report between control block and equipment block

	    "FC_EquipmentReport"(iUDT_Status := #sUDT_CommonStatus,
	                         iqUDT_Control := #iqUDT_EquipmentControl);

	END_REGION

END_FUNCTION_BLOCK

FUNCTION_BLOCK "FB_Conveyor"
TITLE = FB_Conveyor_BiDirectional
{ S7_Optimized_Access := 'TRUE' }
AUTHOR : MHSE
FAMILY : Equimpent
VERSION : 3.0
// ATTRIBUTES
// AUTO_NUMBER = True
// BLOCK_NUMBER = 207
// END_ATTRIBUTES
//Function block to control the bi-directional conveyor.
   VAR_INPUT
      iUDT_ConveyorConfiguration { ExternalAccessible := 'False'; ExternalVisible := 'False'; ExternalWritable := 'False'} : "UDT_ConveyorConfiguration";   //           Conveyor configuration structure
      idi_PECEoSDistance { ExternalAccessible := 'False'; ExternalVisible := 'False'; ExternalWritable := 'False'} : DInt;   //           Distance between photo eye and the end of conveyor [mm] in forward direction
      idi_PECBoSDistance { ExternalAccessible := 'False'; ExternalVisible := 'False'; ExternalWritable := 'False'} : DInt;   //           Distance between photo eye and the end of conveyor [mm] in reverse direction
      ii_ExternalSpeed { ExternalAccessible := 'False'; ExternalVisible := 'False'; ExternalWritable := 'False'} : Int;   //           External speed [mm/s]
      ix_SafetyOk { ExternalAccessible := 'False'; ExternalVisible := 'False'; ExternalWritable := 'False'} : Bool;   //           TRUE when safety is ok
      ix_24vOk { ExternalAccessible := 'False'; ExternalVisible := 'False'; ExternalWritable := 'False'} : Bool;   //           TRUE when 24VDC is healthy
      ix_400vOk { ExternalAccessible := 'False'; ExternalVisible := 'False'; ExternalWritable := 'False'} : Bool;   //           TRUE when 400VAC is healthy
      ix_HardwareOk { ExternalAccessible := 'False'; ExternalVisible := 'False'; ExternalWritable := 'False'} : Bool;   //           TRUE when  hardware is Ok
      ix_PECEoS { ExternalAccessible := 'False'; ExternalVisible := 'False'; ExternalWritable := 'False'} : Bool := TRUE;   //           TRUE when the end of section photoeye in forward direction is not blocked
      ix_PECBoS { ExternalAccessible := 'False'; ExternalVisible := 'False'; ExternalWritable := 'False'} : Bool := TRUE;   //           TRUE when the end of section photoeye in reverse direction is not blocked
      ix_ReverseDirection { ExternalAccessible := 'False'; ExternalVisible := 'False'; ExternalWritable := 'False'} : Bool;   //           FALSE when to run in forward direction and True to run in Reverse direction
      ix_ExternalRequestDieBack { ExternalAccessible := 'False'; ExternalVisible := 'False'; ExternalWritable := 'False'} : Bool;   //           External input to request die back
      ix_ExternalRequestHold { ExternalAccessible := 'False'; ExternalVisible := 'False'; ExternalWritable := 'False'} : Bool;   //           External input to request conveyor hold
      ix_ResetEnergySave { ExternalAccessible := 'False'; ExternalVisible := 'False'; ExternalWritable := 'False'} : Bool;   //           Reset energy save mode timer
   END_VAR

   VAR_OUTPUT
      qUDT_HMIStatus { ExternalAccessible := 'False'; ExternalVisible := 'False'; ExternalWritable := 'False'} : "UDT_ConveyorStatus";   //           HMI status structure
      qUDT_Status { ExternalAccessible := 'False'; ExternalVisible := 'False'; ExternalWritable := 'False'} : "UDT_CommonStatus";   //           Common status structure
   END_VAR

   VAR_IN_OUT
      iqUDT_EquipmentControl : "UDT_EquipmentControl";   //           Equipment control structure
      iqUDT_ConveyorCommand : "UDT_ConveyorCommand";   //           Conveyor command stucture
      iqUDT_ConveyorInterface : "UDT_ConveyorInterface";   //           Interface structure
      iqUDT_HandShakeUp : "UDT_ConveyorHandshake";   //           Upstream handshake structure in forward direction
      iqUDT_HandShake : "UDT_ConveyorHandshake";   //           Handshake structure in forward direction
      iqUDT_Statistics : "UDT_ConveyorStatistics";   //           Statistics structure
   END_VAR

   VAR
      sUDT_CommonStatus { ExternalAccessible := 'False'; ExternalVisible := 'False'; ExternalWritable := 'False'; S7_SetPoint := 'False'} : "UDT_CommonStatus";   //           Common status structure
      sUDT_CommonStatusOld { ExternalAccessible := 'False'; ExternalVisible := 'False'; ExternalWritable := 'False'; S7_SetPoint := 'False'} : "UDT_CommonStatus";   //           Auxiliary status structure
      sUDT_HMIStatus { ExternalAccessible := 'False'; ExternalVisible := 'False'; ExternalWritable := 'False'; S7_SetPoint := 'False'} : "UDT_ConveyorStatus";   //           HMI status structure
      sFB_CascadeModeTimer { ExternalAccessible := 'False'; ExternalVisible := 'False'; ExternalWritable := 'False'; S7_SetPoint := 'False'} : "FB_TimerOnOffDelay";   //           Timer to cascade start
   END_VAR
   VAR RETAIN
      sdi_GapHeadToHeadConfigurationFwd { ExternalAccessible := 'False'; ExternalVisible := 'False'; ExternalWritable := 'False'} : DInt;   //           Preset forward gap head to head with correction [cm]
      sdi_GapTailToHeadConfigurationFwd { ExternalAccessible := 'False'; ExternalVisible := 'False'; ExternalWritable := 'False'} : DInt;   //           Preset forward gap tail to head with correction [cm]
      sdi_GapHeadToHeadConfigurationRvs { ExternalAccessible := 'False'; ExternalVisible := 'False'; ExternalWritable := 'False'} : DInt;   //           Preset reverse gap head to head with correction [cm]
      sdi_GapTailToHeadConfigurationRvs { ExternalAccessible := 'False'; ExternalVisible := 'False'; ExternalWritable := 'False'} : DInt;   //           Preset reverse gap tail to head with correction [cm]
      sdi_AuxGapHeadToHeadCounterFwd { ExternalAccessible := 'False'; ExternalVisible := 'False'; ExternalWritable := 'False'} : DInt;   //           Aux variable to count the head to head
      sdi_AuxGapTailtoHeadCounterFwd { ExternalAccessible := 'False'; ExternalVisible := 'False'; ExternalWritable := 'False'} : DInt;   //           Aux variable to count the gap
      sdi_AuxGapHeadToHeadCounterRvs { ExternalAccessible := 'False'; ExternalVisible := 'False'; ExternalWritable := 'False'} : DInt;   //           Aux variable to count the head to head
      sdi_AuxGapTailtoHeadCounterRvs { ExternalAccessible := 'False'; ExternalVisible := 'False'; ExternalWritable := 'False'} : DInt;   //           Aux variable to count the gap
      sdi_GapFwd { ExternalAccessible := 'False'; ExternalVisible := 'False'; ExternalWritable := 'False'} : DInt;   //           Gap between two products
      sdi_GapHeadToHeadFwd { ExternalAccessible := 'False'; ExternalVisible := 'False'; ExternalWritable := 'False'} : DInt;   //           Head to head between two products
      sdi_Gap_Rvs { ExternalAccessible := 'False'; ExternalVisible := 'False'; ExternalWritable := 'False'} : DInt;   //           Gap between two products
      sdi_GapHeadToHeadRvs { ExternalAccessible := 'False'; ExternalVisible := 'False'; ExternalWritable := 'False'} : DInt;   //           Head to head between two products
      sdi_TailToBeginFwd { ExternalAccessible := 'False'; ExternalVisible := 'False'; ExternalWritable := 'False'} : DInt;   //           Count tail to next conveyor distance
      sdi_HeadToEndFwd { ExternalAccessible := 'False'; ExternalVisible := 'False'; ExternalWritable := 'False'} : DInt;   //           Count head to end distance
      sdi_TailToBeginRvs { ExternalAccessible := 'False'; ExternalVisible := 'False'; ExternalWritable := 'False'} : DInt;   //           Count tail to next conveyor distance
      sdi_HeadToEndRvs { ExternalAccessible := 'False'; ExternalVisible := 'False'; ExternalWritable := 'False'} : DInt;   //           Count head to end distance
      sdi_PECEoSDistanceFwd { ExternalAccessible := 'False'; ExternalVisible := 'False'; ExternalWritable := 'False'} : DInt;   //           Real distance between PEC and the end of distance
      sdi_PECtoEndDistanceFwd { ExternalAccessible := 'False'; ExternalVisible := 'False'; ExternalWritable := 'False'} : DInt;   //           Distance between photeye and the end of the conveyor in cm
      sdi_PEC_EoSDistanceRvs { ExternalAccessible := 'False'; ExternalVisible := 'False'; ExternalWritable := 'False'} : DInt;   //           Real distance between PEC and the end of distance
      sdi_PECtoEndDistanceRvs { ExternalAccessible := 'False'; ExternalVisible := 'False'; ExternalWritable := 'False'} : DInt;   //           Distance between photeye and the end of the conveyor in cm
      sdi_AuxEnergySaveFwd { ExternalAccessible := 'False'; ExternalVisible := 'False'; ExternalWritable := 'False'} : DInt;   //           Auxiliary variable to calculate energy save displacement
      sdi_AuxEnergySaveRvs { ExternalAccessible := 'False'; ExternalVisible := 'False'; ExternalWritable := 'False'} : DInt;   //           Auxiliary variable to calculate energy save displacement
      sdi_DownstreamGapTailtoHeadFwd { ExternalAccessible := 'False'; ExternalVisible := 'False'; ExternalWritable := 'False'} : DInt;   //           Gap between the beginning of the conveyor and the closer parcel in that conveyor
      sdi_DownstreamGapHeadToHeadFwd { ExternalAccessible := 'False'; ExternalVisible := 'False'; ExternalWritable := 'False'} : DInt;   //           Head to head between the beginning of the conveyor and the closer parcel in that conveyor
      sdi_DownstreamGapTailtoHeadRvs { ExternalAccessible := 'False'; ExternalVisible := 'False'; ExternalWritable := 'False'} : DInt;   //           Gap between the beginning of the conveyor and the closer parcel in that conveyor
      sdi_DownstreamGapHeadToHeadRvs { ExternalAccessible := 'False'; ExternalVisible := 'False'; ExternalWritable := 'False'} : DInt;   //           Head to head between the beginning of the conveyor and the closer parcel in that conveyor
      sdi_TransitionZone { ExternalAccessible := 'False'; ExternalVisible := 'False'; ExternalWritable := 'False'} : DInt;   // Counter of product in transition zone
   END_VAR
   VAR
      sR_TRIG_ManualMode {InstructionName := 'R_TRIG'; LibVersion := '1.0'; ExternalAccessible := 'False'; ExternalVisible := 'False'; ExternalWritable := 'False'; S7_SetPoint := 'False'} : R_TRIG;   //           Rising edge trigger manual mode
      sR_TRIG_Jog {InstructionName := 'R_TRIG'; LibVersion := '1.0'; ExternalAccessible := 'False'; ExternalVisible := 'False'; ExternalWritable := 'False'; S7_SetPoint := 'False'} : R_TRIG;   //           Rising edge trigger manual jog
      sR_TRIG_PE_EoSFiltered_Rvs {InstructionName := 'R_TRIG'; LibVersion := '1.0'; ExternalAccessible := 'False'; ExternalVisible := 'False'; ExternalWritable := 'False'; S7_SetPoint := 'False'} : R_TRIG;   //           Rising edge trigger end of section photo eye filtered
      sR_TRIG_PE_EoSFiltered_Fwd {InstructionName := 'R_TRIG'; LibVersion := '1.0'; ExternalAccessible := 'False'; ExternalVisible := 'False'; ExternalWritable := 'False'; S7_SetPoint := 'False'} : R_TRIG;   //           Rising edge trigger end of section photo eye filtered
      sR_TRIG_TailToBegin_Rvs {InstructionName := 'R_TRIG'; LibVersion := '1.0'; ExternalAccessible := 'False'; ExternalVisible := 'False'; ExternalWritable := 'False'; S7_SetPoint := 'False'} : R_TRIG;   //           Rising edge trigger Tail arrive at the beginning of next conveyor
      sR_TRIG_TailToBegin_Fwd {InstructionName := 'R_TRIG'; LibVersion := '1.0'; ExternalAccessible := 'False'; ExternalVisible := 'False'; ExternalWritable := 'False'; S7_SetPoint := 'False'} : R_TRIG;   //           Rising edge trigger Tail arrive at the beginning of next conveyor
      sF_TRIG_ManualMode {InstructionName := 'F_TRIG'; LibVersion := '1.0'; ExternalAccessible := 'False'; ExternalVisible := 'False'; ExternalWritable := 'False'; S7_SetPoint := 'False'} : F_TRIG;   //           Falling edge trigger manual mode
      sF_TRIG_Jog {InstructionName := 'F_TRIG'; LibVersion := '1.0'; ExternalAccessible := 'False'; ExternalVisible := 'False'; ExternalWritable := 'False'; S7_SetPoint := 'False'} : F_TRIG;   //           Falling edge trigger manual mode jog
      sF_TRIG_PEC_EoSFiltered_Rvs {InstructionName := 'F_TRIG'; LibVersion := '1.0'; ExternalAccessible := 'False'; ExternalVisible := 'False'; ExternalWritable := 'False'; S7_SetPoint := 'False'} : F_TRIG;   //           Falling edge trigger end of section photo eye filtered
      sF_TRIG_PEC_EoSFiltered_Fwd {InstructionName := 'F_TRIG'; LibVersion := '1.0'; ExternalAccessible := 'False'; ExternalVisible := 'False'; ExternalWritable := 'False'; S7_SetPoint := 'False'} : F_TRIG;   //           Falling edge trigger end of section photo eye filtered
      sF_TRIG_AuxHeadToEnd_Rvs {InstructionName := 'F_TRIG'; LibVersion := '1.0'; ExternalAccessible := 'False'; ExternalVisible := 'False'; ExternalWritable := 'False'; S7_SetPoint := 'False'} : F_TRIG;   //           Falling edge trigger Aux head to end bit
      sF_TRIG_AuxHeadToEnd_Fwd {InstructionName := 'F_TRIG'; LibVersion := '1.0'; ExternalAccessible := 'False'; ExternalVisible := 'False'; ExternalWritable := 'False'; S7_SetPoint := 'False'} : F_TRIG;   //           Falling edge trigger Aux head to end bit
      sR_TRIG_ConveyorUp {InstructionName := 'R_TRIG'; LibVersion := '1.0'; ExternalAccessible := 'False'; ExternalVisible := 'False'; ExternalWritable := 'False'; S7_SetPoint := 'False'} : R_TRIG;   //           Rising edge trigger conveyor up time
      sR_TRIG_EnergySave {InstructionName := 'R_TRIG'; LibVersion := '1.0'; ExternalAccessible := 'False'; ExternalVisible := 'False'; ExternalWritable := 'False'; S7_SetPoint := 'False'} : R_TRIG;   //           Rising edge trigger energy save
      sR_TRIG_VFDRunning {InstructionName := 'R_TRIG'; LibVersion := '1.0'; ExternalAccessible := 'False'; ExternalVisible := 'False'; ExternalWritable := 'False'; S7_SetPoint := 'False'} : R_TRIG;   //           Rising edge trigger VFD running
      sR_TRIG_ConveyorDownTime {InstructionName := 'R_TRIG'; LibVersion := '1.0'; ExternalAccessible := 'False'; ExternalVisible := 'False'; ExternalWritable := 'False'; S7_SetPoint := 'False'} : R_TRIG;   //           Rising edge trigger conveyor down
      sR_TRIG_RunManual {InstructionName := 'R_TRIG'; LibVersion := '1.0'; ExternalAccessible := 'False'; ExternalVisible := 'False'; ExternalWritable := 'False'; S7_SetPoint := 'False'} : R_TRIG;   //           Rising edge run conveyor in manual mode
      sR_TRIG_Transfering_Rvs {InstructionName := 'R_TRIG'; LibVersion := '1.0'; ExternalAccessible := 'False'; ExternalVisible := 'False'; ExternalWritable := 'False'; S7_SetPoint := 'False'} : R_TRIG;   //           Rising edge transfering
      sR_TRIG_Transfering_Fwd {InstructionName := 'R_TRIG'; LibVersion := '1.0'; ExternalAccessible := 'False'; ExternalVisible := 'False'; ExternalWritable := 'False'; S7_SetPoint := 'False'} : R_TRIG;   //           Rising edge transfering
      sF_TRIG_HeadAtEnd_Rvs {InstructionName := 'F_TRIG'; LibVersion := '1.0'; ExternalAccessible := 'False'; ExternalVisible := 'False'; ExternalWritable := 'False'; S7_SetPoint := 'False'} : F_TRIG;   //           Falling edge head at the end of the conveyor
      sF_TRIG_HeadAtEnd_Fwd {InstructionName := 'F_TRIG'; LibVersion := '1.0'; ExternalAccessible := 'False'; ExternalVisible := 'False'; ExternalWritable := 'False'; S7_SetPoint := 'False'} : F_TRIG;   //           Falling edge head at the end of the conveyor
      sR_TRIG_Reverse {InstructionName := 'R_TRIG'; LibVersion := '1.0'; ExternalAccessible := 'False'; ExternalVisible := 'False'; ExternalWritable := 'False'; S7_SetPoint := 'False'} : R_TRIG;   //           Rising edge of reverse direction
      sF_TRIG_Reverse {InstructionName := 'F_TRIG'; LibVersion := '1.0'; ExternalAccessible := 'False'; ExternalVisible := 'False'; ExternalWritable := 'False'; S7_SetPoint := 'False'} : F_TRIG;   //           Falling edge of reverse direction
      sR_Trig_DirectionChange {InstructionName := 'R_TRIG'; LibVersion := '1.0'; ExternalAccessible := 'False'; ExternalVisible := 'False'; ExternalWritable := 'False'; S7_SetPoint := 'False'} : R_TRIG;   //           Rising edge of change direction
      sF_Trig_DirectionChange {InstructionName := 'F_TRIG'; LibVersion := '1.0'; ExternalAccessible := 'False'; ExternalVisible := 'False'; ExternalWritable := 'False'; S7_SetPoint := 'False'} : F_TRIG;   //           Falling edge of change direction
      sR_TRIG_PrestartManual {InstructionName := 'R_TRIG'; LibVersion := '1.0'; ExternalAccessible := 'False'; ExternalVisible := 'False'; ExternalWritable := 'False'; S7_SetPoint := 'False'} : R_TRIG;   //   Rising edge of manual prestart
      sR_TRIG_ConveyorStopped {InstructionName := 'R_TRIG'; LibVersion := '1.0'; ExternalAccessible := 'False'; ExternalVisible := 'False'; ExternalWritable := 'False'; S7_SetPoint := 'False'} : R_TRIG;   //  Rising edge of stop
      sx_Ready { ExternalAccessible := 'False'; ExternalVisible := 'False'; ExternalWritable := 'False'} : Bool;   //           Conveyor Ready to operate in Automatic mode
   END_VAR
   VAR RETAIN
      sx_StartReceived { ExternalAccessible := 'False'; ExternalVisible := 'False'; ExternalWritable := 'False'} : Bool;   //           Save start trigger from the system
      sx_EnergySaveActive { ExternalAccessible := 'False'; ExternalVisible := 'False'; ExternalWritable := 'False'} : Bool;   //           Active energy save mode
      sx_AuxHeadToEndFwd { ExternalAccessible := 'False'; ExternalVisible := 'False'; ExternalWritable := 'False'} : Bool;   //           Aux bit to control head to end positioning in forward direction
      sx_AuxHeadToEndRvs { ExternalAccessible := 'False'; ExternalVisible := 'False'; ExternalWritable := 'False'} : Bool;   //           Aux bit to control head to end positioning in reverse direction
      sx_TailToBeginFwd { ExternalAccessible := 'False'; ExternalVisible := 'False'; ExternalWritable := 'False'} : Bool;   //           Tail to begin done in forward direction
      sx_TailToBeginRvs { ExternalAccessible := 'False'; ExternalVisible := 'False'; ExternalWritable := 'False'} : Bool;   //           Tail to begin done in reverse direction
      sx_GappingFwd { ExternalAccessible := 'False'; ExternalVisible := 'False'; ExternalWritable := 'False'} : Bool;   //           Gapping in process in forward direction
      sx_GappingRvs { ExternalAccessible := 'False'; ExternalVisible := 'False'; ExternalWritable := 'False'} : Bool;   //           Gapping in process in reverse direction
   END_VAR
   VAR
      sx_AutomaticActive { ExternalAccessible := 'False'; ExternalVisible := 'False'; ExternalWritable := 'False'} : Bool;   //           Automatic active
   END_VAR
   VAR RETAIN
      sx_RecoveryGapFwd { ExternalAccessible := 'False'; ExternalVisible := 'False'; ExternalWritable := 'False'} : Bool;   //           Recovery gap activated in forward direction
      sx_RecoveryGapRvs { ExternalAccessible := 'False'; ExternalVisible := 'False'; ExternalWritable := 'False'} : Bool;   //           Recovery gap activated in reverse direction
   END_VAR
   VAR
      sx_ManualModeActive { ExternalAccessible := 'False'; ExternalVisible := 'False'; ExternalWritable := 'False'} : Bool;   //           Manual mode active
      sx_PreStartManual { ExternalAccessible := 'False'; ExternalVisible := 'False'; ExternalWritable := 'False'} : Bool;   //           Pre conditions to run conveyor in manual mode
   END_VAR
   VAR RETAIN
      sx_AuxHeadAtEndFwd { ExternalAccessible := 'False'; ExternalVisible := 'False'; ExternalWritable := 'False'} : Bool;   //           Parcel reach the end of the conveyor in forward direction
      sx_AuxHeadAtEndRvs { ExternalAccessible := 'False'; ExternalVisible := 'False'; ExternalWritable := 'False'} : Bool;   //           Parcel reach the end of the conveyor in reverse direction
   END_VAR
   VAR
      sx_CascadeStartUp { ExternalAccessible := 'False'; ExternalVisible := 'False'; ExternalWritable := 'False'} : Bool;   //           Cascade startup auxiliary bit
      sx_DirectionChanged { ExternalAccessible := 'False'; ExternalVisible := 'False'; ExternalWritable := 'False'} : Bool;   //           Change direction until stop
      sx_ReverseDirection { ExternalAccessible := 'False'; ExternalVisible := 'False'; ExternalWritable := 'False'} : Bool;   //           Direction Selection auxiliary bit
      sx_ManualRunning { ExternalAccessible := 'False'; ExternalVisible := 'False'; ExternalWritable := 'False'} : Bool;   //          Conveyor running in manual mode
      sx_Up { ExternalAccessible := 'False'; ExternalVisible := 'False'; ExternalWritable := 'False'} : Bool;   //  Conveyor is up
      sx_Down { ExternalAccessible := 'False'; ExternalVisible := 'False'; ExternalWritable := 'False'} : Bool;   //  Conveyor is down
      sx_Stopped { ExternalAccessible := 'False'; ExternalVisible := 'False'; ExternalWritable := 'False'} : Bool;   //  Conveyor is stopped
   END_VAR

   VAR_TEMP
      tx_CascadeStart : Bool;
   END_VAR

   VAR CONSTANT
      ci_OverflowLimit : Int := 32000;   //           Limit int overflow
   END_VAR


BEGIN
	(*
	----------------------------------------------------------------------------------------

	Version history:
	Date        | Version   | Author        | Remark
	----------------------------------------------------------------------------------------
	            | 3.0       | C.Leite       | First release TIA 15.1
	01/01/2020  | 3.1       | S. Deulkar    | Modified error loging, added reset to reset internal error
	                                        | Cosidered commissioning error to put conveyor in ready state
	07/01/2020  | 3.2       | C. Leite      | Manual mode bug corrected related with conveyor start
	10/01/2020  | 3.3       | C. Leite      | Manual mode start\stop change
	                                        | Lenght conveyor data type was changed to DInt
	14/01/2020  | 3.4       | F.Baten       | Renamed Trail to Tail
	                                        | Renamed ii_PEC_EosDistance_EoS to idi_PEC_EoSDistance same for BoS
	21/01/2020  | 3.5       | C.Leite       | Reset gapping bits when the direction changes
	06/01/2020  | 3.6       | S. Deulkar    | Added safety Ok in condition to make ready status
	25/02/2020  | 3.7       | S. Deulkar    | Modified to update ststus output every cycle
	21/04/2020  | 3.8       | F.Baten       | Modified energysave reset
	23/04/2020  | 3.9       | S. Deulkar    | Modified logic for reset energy save command if it is slave conveyor
	22/06/2020  | 3.10      | K. Pokorski   | Modified singaling request activation, modified stop conditions (Handshake ReqStop)
	02/07/2020  | 3.11      | K. Pokorski   | Modified condition to disable manual mode (safety ok)
	30/07/2020  | 3.12      | S. Theocharis | Reset HMI commands of manual mode when conveyor no ready
	                                        | Keep downstream running when the a PEC error occurs
	04/08/2020  | 3.13      | S. Deulkar    | Deletded Manual run stop command and Modified code to let
	                                        | let slave conveyor go in energy save, Optimized energy save logic
	17/08/2020  | 3.14      | L.Klar        | Gapping corrected to work with PEC offset. Gap correction configuration added
	17/08/2020  | 3.15      | S. Theocharis | Encoder fault added. Manual mode active to interface. Stop trigger added for statistics
	                                        | Fix  statistics
	11/01/2021  | 3.16      | L.Klar        | Input safety ok added to stop conveyor condition
	02/03/2021  | 3.17      | K. Pokorski   | Halted status enable only when automatic on
	11/03/2021  | 3.18      | S. Theocharis | Added bulk flow mode 3
	13/03/2021  | 3.19      | S. Theocharis | Warning color commented, line 665 added, sensors initial values changed to true
	15/03/2021  | 3.20      | S. Theocharis | Energy safe corrected
	29/03/2021  | 3.21      | M. Kocot      | Added HMI command for manual speed percetage selection and modified logic for cascade
	                                        | startup
	31/03/2021  | 3.22      | H.Rutkowski   | Changed logic for TransitionZone calculation in mode 3( Converted PEC distance to cm)
	14/05/2021  | 3.23      | S. Nikodem    | Reset value from iq_UDT_HandShakeUp.DownstreamDisplacement and iq_UDT_HandShake.DownstreamDisplacement
	28/06/2021  | 3.24      | N.Kadam       | Modified logic for conveyor downtime and Esave statistics
	29/07/2021  | 3.25      | S. Deulkar    | Autotic ON condition is added to excecut region 7: Automatic mode active
	                                        | Statistics are updated after status
	11/11/2021  | 3.26      | M.Singh       |Shared Hardware signal over Interface
	28/03/2022  | 3.27      | M.Singh       |Solved Esave Bug, Swapped regions "Operation modes" and "Energy Save"
	28/07/2022  | 3.28      | M.Singh       |Removed handsakeUP.RTR from conditions determining downstream TIP and RTS
	30/07/2022  | 3.28      | M.Singh       |Addded hardware ok as condition to show safety status
	                                        |Added Aux Head at end and TIP to Esave Reset conditions


	*)

	REGION 1 - Initial

	    REGION 1.1 - First PLC cycle

	        // Conveyor stops in the first scan of the PLC
	        IF "DB_Memory".FirstScan
	        THEN
	            #iqUDT_EquipmentControl.Command.Start := FALSE;    // Command start
	            #sx_AutomaticActive := FALSE;                       // switch of automatic active
	            #iqUDT_HandShakeUp.RTR := False;                   // Reset RTR signal

	            #iqUDT_HandShakeUp.CascadeStartUp := FALSE;        // Reset cascade start signal

	            #iqUDT_ConveyorInterface.RunFwd := FALSE;          // Order to run forward to VFD
	            #iqUDT_ConveyorInterface.RunRvs := FALSE;          // Order to run reverse to VFD

	        END_IF;

	    END_REGION

	    REGION 1.2 - Conversion distance between PEC and end of conveyor [mm to cm]

	        // Move PEC Distance into a static variable. Added on version 2.8
	        #sdi_PECEoSDistanceFwd := #idi_PECEoSDistance;
	        #sdi_PEC_EoSDistanceRvs := #iUDT_ConveyorConfiguration.Common.Length - #idi_PECBoSDistance;

	        // Limit to prevent malfunctions with zero or negative values. Added on version 2.8
	        IF #sdi_PECEoSDistanceFwd < 10
	        THEN
	            #sdi_PECEoSDistanceFwd := 10;
	        END_IF;

	        IF #sdi_PEC_EoSDistanceRvs < 10
	        THEN
	            #sdi_PEC_EoSDistanceRvs := 10;
	        END_IF;

	        //  Convertion of the distance between photo eye and the end of the conveyor from mm to cm.
	        #sdi_PECtoEndDistanceFwd := (#sdi_PECEoSDistanceFwd
	        - #iUDT_ConveyorConfiguration.Forward_Direction.PEC_EoSDistanceOffset) / 10;

	        #sdi_PECtoEndDistanceRvs := (#sdi_PEC_EoSDistanceRvs
	        - #iUDT_ConveyorConfiguration.Reverse_Direction.PEC_BoSDistanceOffset) / 10;


	        // Limit the Pec to End distance in positive ranges. Added on version 2.7
	        IF #sdi_PECtoEndDistanceFwd < 1 THEN
	            #sdi_PECtoEndDistanceFwd := 1;
	        END_IF;

	        IF #sdi_PECtoEndDistanceRvs < 1 THEN
	            #sdi_PECtoEndDistanceRvs := 1;
	        END_IF;

	        #sx_ReverseDirection := (#iqUDT_ConveyorCommand.Reverse OR #ix_ReverseDirection) AND #iUDT_ConveyorConfiguration.Bi_Directional_Enable;


	    END_REGION

	    REGION 1.3 Conditions Up - Down - Stopped
	        //Used for statistics

	        #sx_Up := (#sx_AutomaticActive                               // Automatic active
	        AND #sx_Ready                                                // Ready active
	        AND NOT #sx_EnergySaveActive);                              // Not in energy save

	        #sx_Down := (NOT #sx_ManualModeActive                                                   // Not in manual mode
	        AND #sUDT_CommonStatus.Error                                                           // in error
	        AND NOT #sx_Ready                                                                       // Conveyor not ready
	        AND NOT #sx_EnergySaveActive);                                                          // Not in energy save

	        #sx_Stopped := (NOT #sx_AutomaticActive AND #sx_Ready);

	    END_REGION

	    REGION 1.3 - Triggers

	        // Rising edge trigger manual mode
	        #sR_TRIG_ManualMode(CLK := #iqUDT_ConveyorCommand.ManualMode
	                            OR #iqUDT_EquipmentControl.Command.ManualMode);

	        // Falling edge trigger manual mode
	        #sF_TRIG_ManualMode(CLK := #iqUDT_ConveyorCommand.ManualMode
	                            OR #iqUDT_EquipmentControl.Command.ManualMode);

	        // Rising edge trigger manual mode jog
	        #sR_TRIG_Jog(CLK := #iqUDT_ConveyorCommand.ManualJog);

	        // Falling edge trigger manual mode jog
	        #sF_TRIG_Jog(CLK := #iqUDT_ConveyorCommand.ManualJog);

	        // Rising edge trigger to start in manual mode
	        #sR_TRIG_RunManual(CLK := #iqUDT_ConveyorCommand.ManualStartStop);

	        // Rising edge trigger end of section photo eye filtered
	        #sR_TRIG_PE_EoSFiltered_Fwd(CLK := #ix_PECEoS);
	        #sR_TRIG_PE_EoSFiltered_Rvs(CLK := #ix_PECBoS);

	        // Falling edge trigger end of section photo eye filtered
	        #sF_TRIG_PEC_EoSFiltered_Fwd(CLK := #ix_PECEoS);
	        #sF_TRIG_PEC_EoSFiltered_Rvs(CLK := #ix_PECBoS);

	        // Rising edge conveyor up
	        #sR_TRIG_ConveyorUp(CLK := #sx_Up);

	        // Rising edge energy save mode
	        #sR_TRIG_EnergySave(CLK := #sx_EnergySaveActive);

	        // Rising edge running
	        #sR_TRIG_VFDRunning(CLK := #iqUDT_ConveyorInterface.VFDRunning);

	        // Rising edge conveyor conveyor down
	        #sR_TRIG_ConveyorDownTime(CLK := #sx_Down);

	        //Rising edge conveyor stopped
	        #sR_TRIG_ConveyorStopped(CLK := #sx_Stopped);

	        // Rising edge conveyor command reverse direction
	        #sR_TRIG_Reverse(CLK := #iqUDT_ConveyorCommand.Reverse);

	        // Falling edge conveyor command reverse direction
	        #sF_TRIG_Reverse(CLK := #iqUDT_ConveyorCommand.Reverse);

	        // Rising edge conveyor change direction
	        #sR_Trig_DirectionChange(CLK := #sx_ReverseDirection);

	        // Falling edge conveyor change direction
	        #sF_Trig_DirectionChange(CLK := #sx_ReverseDirection);

	    END_REGION

	    REGION 1.4 - Move displacement to upstream

	        // Downstream displacement is mode to upstream conveyor to calculate gap

	        IF NOT #sx_ReverseDirection
	        THEN
	            #iqUDT_HandShakeUp.DownstreamDisplacement := #iqUDT_ConveyorInterface.Displacement;
	        ELSE
	            #iqUDT_HandShake.DownstreamDisplacement := #iqUDT_ConveyorInterface.Displacement;

	        END_IF;

	    END_REGION

	    REGION 1.5 - Change direction

	        // The memory bit to change direction is activated when the input is trigger

	        IF #sR_Trig_DirectionChange.Q
	            OR #sF_Trig_DirectionChange.Q
	        THEN
	            #sx_DirectionChanged := TRUE;
	        END_IF;

	        // The direction changed memory bit is just reset when the conveyor stops to prevente mechanical problems

	        IF #sx_DirectionChanged
	            AND #iUDT_ConveyorConfiguration.Bi_Directional_Enable
	            AND NOT #iqUDT_ConveyorInterface.VFDatSpeed
	            AND NOT #iqUDT_ConveyorInterface.VFDRunning
	            AND (#iqUDT_ConveyorInterface.ActualSpeed <= 0)
	        THEN
	            #sx_DirectionChanged := FALSE;

	            #sx_AuxHeadAtEndFwd := FALSE;
	            #sx_AuxHeadAtEndRvs := FALSE;

	            #sdi_AuxGapHeadToHeadCounterFwd := 0;
	            #sdi_AuxGapHeadToHeadCounterRvs := 0;

	            #sdi_AuxGapTailtoHeadCounterRvs := 0;
	            #sdi_AuxGapTailtoHeadCounterFwd := 0;

	            #sx_GappingRvs := FALSE;
	            #sx_GappingFwd := FALSE;

	            #iqUDT_HandShake.TIP := FALSE;
	            #iqUDT_HandShakeUp.TIP := FALSE;

	            #iqUDT_HandShakeUp.DownstreamDisplacement := 0;     // v3.23
	            #iqUDT_HandShake.DownstreamDisplacement := 0;       // v3.23

	        END_IF;

	        IF (#sR_Trig_DirectionChange.Q
	            AND NOT #ix_PECBoS)
	            OR (#sF_Trig_DirectionChange.Q
	            AND NOT #ix_PECEoS)
	            AND #iUDT_ConveyorConfiguration.Bi_Directional_Enable
	        THEN
	            #sdi_AuxGapHeadToHeadCounterFwd := 0;
	            #sdi_AuxGapHeadToHeadCounterRvs := 0;
	        END_IF;

	    END_REGION

	    REGION 1.5 - Gaps configuration

	        // Forward head to head
	        #sdi_GapHeadToHeadConfigurationFwd := #iUDT_ConveyorConfiguration.Forward_Direction.GapHeadToHead + #iUDT_ConveyorConfiguration.Forward_Direction.GapCorrection;
	        // Forward tail to head
	        #sdi_GapTailToHeadConfigurationFwd := #iUDT_ConveyorConfiguration.Forward_Direction.GapTailToHead + #iUDT_ConveyorConfiguration.Forward_Direction.GapCorrection;
	        // Reverse head to head
	        #sdi_GapHeadToHeadConfigurationRvs := #iUDT_ConveyorConfiguration.Reverse_Direction.GapHeadToHead + #iUDT_ConveyorConfiguration.Reverse_Direction.GapCorrection;
	        // Reverse tail to head
	        #sdi_GapTailToHeadConfigurationRvs := #iUDT_ConveyorConfiguration.Reverse_Direction.GapTailToHead + #iUDT_ConveyorConfiguration.Reverse_Direction.GapCorrection;

	    END_REGION

	END_REGION

	REGION 2 - Reset faults

	    REGION 2.1 - Send reset request to interface UDT

	        // Reset signal is sent to the interface UDT (VFD block, Tracking block, PEC update block)
	        #iqUDT_ConveyorInterface.InternalErrorReset := #iqUDT_EquipmentControl.Command.Reset;

	        #iqUDT_ConveyorInterface.ResetStatistics := #iqUDT_EquipmentControl.Command.ResetData;

	    END_REGION


	    REGION 2.2 - Error / warning

	        #sUDT_CommonStatus.Error := #iqUDT_ConveyorInterface.InternalErrorPEC               // Internal PEC error status
	        OR #iqUDT_ConveyorInterface.InternalErrorVFD               // Internal VFD error status
	        OR #iqUDT_ConveyorInterface.InternalErrorTracking          // Internal tracking error status
	        OR #iqUDT_ConveyorInterface.Disconnected                   // Isolator switch error status
	        OR #iqUDT_ConveyorInterface.InternalErrorEncoder;          // Encoder error


	        #sUDT_CommonStatus.Warning := #iqUDT_ConveyorInterface.InternalWarningTracking        // v2.3 Internal Warning Tracking  added
	        OR #iqUDT_ConveyorInterface.InternalWarningVFD;                                        // v2.3 Internal Warning VFD added

	    END_REGION

	END_REGION

	REGION 3 - Check conditions to set conveyor ready
	    //Share HardwareOK signal over interface
	    #iqUDT_ConveyorInterface.HardwareOk := #ix_HardwareOk;

	    //  Conditions to set bit sx_Ready to operate in automatic mode
	    #sx_Ready := NOT #sUDT_CommonStatus.Error                              // Ready bit is set true when common error status its false
	    AND #ix_SafetyOk
	    AND #ix_24vOk                                                        // 24V error status
	    AND #ix_400vOk                                                       // 400V error status
	    AND #ix_HardwareOk                                                   // Profinet error status
	    AND NOT #iqUDT_ConveyorInterface.ConfigurationError;                // No configuration error

	END_REGION

	REGION 4 - Stop conveyor

	    // Conditions to stop conveyor
	    IF (#sF_TRIG_Jog.Q                                           // Trigger when conveyor stops jogging by HMI
	        AND #sx_ManualModeActive)                                   // Manual mode is active

	        OR (NOT #iqUDT_EquipmentControl.Command.AutomaticOn        // Conveyor stops if the bit AutomaticOn from control block is false
	        AND NOT #sx_ManualModeActive)                               // Manual mode active bit

	        OR (NOT #sx_Ready                                           // Bit conveyor ready to run in automatic mode
	        AND NOT #sx_ManualModeActive)                               // Manual mode active

	        OR #sR_TRIG_ManualMode.Q                                     // Trigger when manual mode is set on
	        OR #sF_TRIG_ManualMode.Q                                     // Trigger when manual mode is set off

	        OR (#iqUDT_HandShakeUp.ReqStop                             // Stop request from upstream if direction not changed
	        AND NOT #sx_DirectionChanged)

	        OR (#iqUDT_HandShake.ReqStop                               // Stop request from downstream if direction changed
	        AND #sx_DirectionChanged)

	        OR NOT #ix_SafetyOk

	    THEN
	        //  Order to stop VFD
	        #iqUDT_ConveyorInterface.RunFwd := FALSE;                  // Set false order to VFD run in forward direction
	        #iqUDT_ConveyorInterface.RunRvs := FALSE;                  // Set false order to VFD run in reverse direction

	        IF NOT #sx_ReverseDirection
	        THEN

	            #iqUDT_HandShakeUp.RTR := FALSE;                       // Set false the bit ready to receive
	            #iqUDT_HandShakeUp.CascadeStartUp := FALSE;            // Set false cascade start up bit

	        ELSE

	            #iqUDT_HandShake.RTR := FALSE;                       // Set false the bit ready to receive
	            #iqUDT_HandShake.CascadeStartUp := FALSE;            // Set false cascade start up bit

	        END_IF;

	        #sx_AutomaticActive := FALSE;                               // Automatic mode is disable
	        //    #sx_StartReceived := FALSE;                                 // Clear start receive bit

	    END_IF;

	END_REGION

	REGION 5 - Start

	    REGION 5.1 - Save Start bit request

	        // The conditions to set the bit "startReceived" are:
	        // - Conveyor not in manual mode.
	        // - Conveyor ready to run.
	        // - Bit AutomaticOn from control block must be on.
	        // - Bit start form control block on.

	        IF #iqUDT_EquipmentControl.Command.Start
	            AND #iqUDT_EquipmentControl.Command.AutomaticOn
	        THEN
	            #sx_StartReceived := TRUE;          // Start bit from control block received
	        END_IF;

	    END_REGION

	    REGION 5.2 - Cascade mode

	        (* If the bit "StartReceived" is set, automatic mode is activated if the conveyor is set as the first one to run
	         or the bit cascadestartup from downstream is on. *)

	        IF #iqUDT_EquipmentControl.Command.Start
	            AND #iqUDT_EquipmentControl.Command.AutomaticOn
	            AND NOT #sx_ManualModeActive
	            AND #sx_Ready
	        THEN
	            #sx_AutomaticActive := TRUE;        // Conveyor active automatic mode
	        END_IF;

	        //Timer to cascade mode
	        #tx_CascadeStart := #sx_StartReceived
	        AND ((NOT #sx_ReverseDirection
	        AND (#iUDT_ConveyorConfiguration.Forward_Direction.FirstConveyorToStart
	        OR #iqUDT_HandShake.CascadeStartUp))
	        OR (#sx_ReverseDirection
	        AND (#iUDT_ConveyorConfiguration.Reverse_Direction.FirstConveyorToStart
	        OR #iqUDT_HandShakeUp.CascadeStartUp)));

	        #sFB_CascadeModeTimer(iudi_OnDelayTime := #iUDT_ConveyorConfiguration.CascadeTimeOnDelay,      // Cascade mode timer
	                              ix_SignalToDelay := #tx_CascadeStart,
	                              ix_Enable := TRUE,                                                   // Signal ready to enable cascade mode
	                              qx_DelayedSignal => #sx_CascadeStartUp);

	        IF NOT #iqUDT_EquipmentControl.Command.AutomaticOn
	        THEN
	            #sx_StartReceived := False;
	        END_IF;


	        // Cascade mode signal to upstream
	        IF NOT #sx_ReverseDirection
	        THEN
	            #iqUDT_HandShakeUp.CascadeStartUp := #sx_CascadeStartUp;
	        ELSE
	            #iqUDT_HandShake.CascadeStartUp := #sx_CascadeStartUp;
	        END_IF;



	    END_REGION

	END_REGION

	REGION 6 - Manual mode

	    REGION 6.1 - Manual mode force disable

	        // Manual mode bits inputs can be reset in case of malfunction
	        IF #iqUDT_EquipmentControl.Command.DisableManualMode
	        THEN
	            #iqUDT_ConveyorCommand.ManualMode := False;
	            #iqUDT_EquipmentControl.Command.ManualMode := False;
	        END_IF;

	    END_REGION

	    REGION 6.2 - Manual mode activation

	        // Manual mode is active if it is active from hmi or by control block
	        #sx_ManualModeActive := #iqUDT_ConveyorCommand.ManualMode
	        OR #iqUDT_EquipmentControl.Command.ManualMode;

	        //Send manual mode active to PEC/VFD blocks to supress errors
	        #iqUDT_ConveyorInterface.ManualModeActive := #sx_ManualModeActive;

	    END_REGION

	    REGION 6.3 - Reset manual commands
	        //When the system is not any more in manual mode or when fatal error occurs the HMI commands should be reset
	        //Added in V3.12 as bug fix.
	        IF NOT #ix_SafetyOk
	            OR NOT #ix_24vOk                                                        // 24V error status
	            OR NOT #ix_400vOk                                                       // 400V error status
	            OR NOT #ix_HardwareOk                                                   // Profinet error status
	            OR #iqUDT_ConveyorInterface.ConfigurationError                          // No configuration err
	            OR #iqUDT_ConveyorInterface.InternalErrorVFD
	            OR #iqUDT_ConveyorInterface.Disconnected
	            OR NOT #sx_ManualModeActive
	        THEN
	            #iqUDT_ConveyorCommand.ManualStartStop := FALSE;
	            #iqUDT_ConveyorCommand.ManualFullSpeed := FALSE;
	            #iqUDT_ConveyorCommand.ManualJog := FALSE;
	            #iqUDT_ConveyorCommand.Reverse := FALSE;
	        END_IF;

	    END_REGION

	    REGION 6.4 - Start/Stop

	        // Pre start conditions to run in manual mode
	        #sx_PreStartManual := #sx_ManualModeActive              // Manual mode active bit
	        AND #ix_SafetyOk                                        // Safety healthy bit
	        AND NOT #iqUDT_ConveyorInterface.Disconnected          // Isolator switch connected
	        AND #ix_HardwareOk                                      // Profinet comunication
	        AND NOT #iqUDT_ConveyorInterface.InternalErrorVFD;     // Internal error from VFD

	        #sR_TRIG_PrestartManual(CLK := #sx_PreStartManual);


	        IF (#sx_PreStartManual                                  // Pre start conditions to run in manual mode
	            AND (#sR_TRIG_RunManual.Q                            // Trigger when conveyor start running in manual mode
	            OR (#iqUDT_ConveyorCommand.ManualStartStop             // Conveyor start running in manual mode active
	            AND #sR_TRIG_PrestartManual.Q)                       // Trigger when pre start conditions ti run in manual mode
	            AND NOT #iqUDT_ConveyorCommand.ManualJog)          // Conveyor is not running in jog
	            OR (#sx_PreStartManual AND #sR_TRIG_Jog.Q                                   // Trigger to start jogging
	            AND NOT #iqUDT_ConveyorCommand.ManualStartStop))       // Conveyor is not running in manual mode
	        THEN

	            #iqUDT_EquipmentControl.Request.SignalingRequest := TRUE;  // Request signaling to control block before conveyor run in manual mode

	        END_IF;

	        // Run conveyor forward in manual mode
	        #iqUDT_ConveyorInterface.RunFwd := #sx_PreStartManual           // Pre start conditions to run in manual mode
	        AND NOT #iqUDT_ConveyorCommand.Reverse                          // Not in reverse direction
	        AND (NOT #iqUDT_EquipmentControl.Request.SignalingRequest       // Signaling request done
	        OR #sx_ManualRunning)
	        AND (#iqUDT_ConveyorCommand.ManualStartStop                         // Manual mode start to run
	        OR #iqUDT_ConveyorCommand.ManualJog);                           // Jogging

	        // Run conveyor reverse in manual mode
	        #iqUDT_ConveyorInterface.RunRvs := #sx_PreStartManual           // Pre start conditions to run in manual mode
	        AND #iqUDT_ConveyorCommand.Reverse                              // Reverse direction
	        AND (NOT #iqUDT_EquipmentControl.Request.SignalingRequest       // Signaling request done
	        OR #sx_ManualRunning)
	        AND (#iqUDT_ConveyorCommand.ManualStartStop                         // Manual mode start to run
	        OR #iqUDT_ConveyorCommand.ManualJog);                           // Jogging

	        #sx_ManualRunning := #iqUDT_ConveyorInterface.RunFwd
	        OR #iqUDT_ConveyorInterface.RunRvs;

	    END_REGION

	END_REGION

	REGION 7 - Automatic mode active

	    IF NOT #sx_ManualModeActive // Manual mode is not active
	    THEN
	        REGION 7.1 - Head to End

	            (*  Function to calculate when the head of the parcel reaches the end of the conveyor
	                When PEC detects parcels head, the functionality increments the displacement of the conveyor until reach the value of the distance
	                between PEC and the end of the conveyor. After that, the counter is reset and the bit #sx_AuxHeadToEnd is triggered to inform the system. *)
	            IF NOT #sx_ReverseDirection
	            THEN
	                REGION 7.1.1 - Forward

	                    IF #sF_TRIG_PEC_EoSFiltered_Fwd.Q      // Detects the product's head
	                    THEN

	                        #sdi_HeadToEndFwd := #sdi_PECtoEndDistanceFwd;                // move the distance between PE and the end of the conveyor to auxiliary variable
	                        #sx_AuxHeadToEndFwd := TRUE;                             // Active head to end function

	                        #sdi_GapHeadToHeadFwd := #sdi_AuxGapHeadToHeadCounterFwd;     // Move gap calculated to variable
	                        #sdi_AuxGapHeadToHeadCounterFwd := 0;                     // Reset gap counter

	                        #sdi_GapFwd := #sdi_AuxGapTailtoHeadCounterFwd;    // Move gap calculated to variable
	                        #sdi_AuxGapTailtoHeadCounterFwd := 0;                     // Reset gap counter

	                        #iqUDT_HandShake.RTS := TRUE;                         // Set ready to send true when a parcel is detected in the PEC

	                    END_IF;

	                    IF #sx_AuxHeadToEndFwd                 // Parcel's head detected in photo cell
	                        AND (#sdi_HeadToEndFwd > 0)         // Psrcel's head do not arrive in the end of the conveyor yet
	                    THEN

	                        #sdi_HeadToEndFwd -= #iqUDT_ConveyorInterface.Displacement;   // Count displacement until arrive to the end of the conveyor

	                    ELSE

	                        #sx_AuxHeadToEndFwd := FALSE;      // Stop function head to end

	                    END_IF;

	                    // Falling edge trigger Aux Head to End bit
	                    #sF_TRIG_AuxHeadToEnd_Fwd(CLK := #sx_AuxHeadToEndFwd);

	                    IF #sF_TRIG_AuxHeadToEnd_Fwd.Q
	                    THEN
	                        #sx_AuxHeadAtEndFwd := TRUE;                       // The head of the parcel is at the front positon of the conveyor
	                    END_IF;


	                    #sF_TRIG_HeadAtEnd_Fwd(CLK := #sx_AuxHeadAtEndFwd);

	                END_REGION
	            ELSE
	                REGION 7.1.2 - Reverse

	                    IF #sF_TRIG_PEC_EoSFiltered_Rvs.Q      // Detects the product's head
	                    THEN

	                        #sdi_HeadToEndRvs := #sdi_PECtoEndDistanceRvs;                // move the distance between PE and the end of the conveyor to auxiliary variable
	                        #sx_AuxHeadToEndRvs := TRUE;                             // Active head to end function

	                        #sdi_GapHeadToHeadRvs := #sdi_AuxGapHeadToHeadCounterRvs;     // Move gap calculated to variable
	                        #sdi_AuxGapHeadToHeadCounterRvs := 0;                     // Reset gap counter

	                        #sdi_Gap_Rvs := #sdi_AuxGapTailtoHeadCounterRvs;    // Move gap calculated to variable
	                        #sdi_AuxGapTailtoHeadCounterRvs := 0;                     // Reset gap counter

	                        #iqUDT_HandShakeUp.RTS := TRUE;                         // Set ready to send true when a parcel is detected in the PEC

	                    END_IF;

	                    IF #sx_AuxHeadToEndRvs                 // Parcel's head detected in photo cell
	                        AND (#sdi_HeadToEndRvs > 0)         // Psrcel's head do not arrive in the end of the conveyor yet
	                    THEN

	                        #sdi_HeadToEndRvs += #iqUDT_ConveyorInterface.Displacement;   // Count displacement until arrive to the end of the conveyor

	                    ELSE

	                        #sx_AuxHeadToEndRvs := FALSE;      // Stop function head to end

	                    END_IF;

	                    // Falling edge trigger Aux Head to End bit
	                    #sF_TRIG_AuxHeadToEnd_Rvs(CLK := #sx_AuxHeadToEndRvs);

	                    IF #sF_TRIG_AuxHeadToEnd_Rvs.Q
	                    THEN
	                        #sx_AuxHeadAtEndRvs := TRUE;                       // The head of the parcel is at the front positon of the conveyor
	                    END_IF;


	                    #sF_TRIG_HeadAtEnd_Rvs(CLK := #sx_AuxHeadAtEndRvs);

	                END_REGION
	            END_IF;
	        END_REGION

	        REGION 7.2 - Tail to Begin

	            (*   This function tracks when parcels tail reaches the begin of downstream conveyor
	                 When the PEC is clear, the function start to increase the displacement until reaches the distance
	                 between PEC and the end of conveyor. *)
	            IF NOT #sx_ReverseDirection
	            THEN
	                REGION 7.2.1 - Forward

	                    IF #sR_TRIG_PE_EoSFiltered_Fwd.Q                     // Detects product's tail
	                    THEN

	                        #sdi_TailToBeginFwd := (#sdi_PECEoSDistanceFwd / 10);   // move distance between PE and the end of the conveyor to auxiliar variable

	                    END_IF;

	                    IF (#sdi_TailToBeginFwd > 0)                                           // While tails parcel do not reach the beginning of next conveyor
	                    THEN

	                        #sdi_TailToBeginFwd -= #iqUDT_ConveyorInterface.Displacement;   // count displacement until the product's tail arrive to the next conveyor
	                        #sx_TailToBeginFwd := FALSE;                                    // Reset tail to begin bit

	                    ELSE

	                        #sx_TailToBeginFwd := TRUE;                                     // Product's tail arrived at the begin OF next conveyor

	                    END_IF;

	                    // Rising edge trigger Aux tail to Begin bit
	                    #sR_TRIG_TailToBegin_Fwd(CLK := #sx_TailToBeginFwd);

	                END_REGION
	            ELSE
	                REGION 7.2.2 - Reverse

	                    IF #sR_TRIG_PE_EoSFiltered_Rvs.Q                     // Detects product's tail
	                    THEN

	                        #sdi_TailToBeginRvs := (#sdi_PEC_EoSDistanceRvs / 10);   // move distance between PE and the end of the conveyor to auxiliar variable

	                    END_IF;

	                    IF (#sdi_TailToBeginRvs > 0)                                           // While tails parcel do not reach the beginning of next conveyor
	                    THEN

	                        #sdi_TailToBeginRvs += #iqUDT_ConveyorInterface.Displacement;   // count displacement until the product's tail arrive to the next conveyor
	                        #sx_TailToBeginRvs := FALSE;                                    // Reset tail to begin bit

	                    ELSE

	                        #sx_TailToBeginRvs := TRUE;                                     // Product's tail arrived at the begin OF next conveyor

	                    END_IF;

	                    // Rising edge trigger Aux tail to Begin bit
	                    #sR_TRIG_TailToBegin_Rvs(CLK := #sx_TailToBeginRvs);

	                END_REGION
	            END_IF;
	        END_REGION

	        REGION 7.3 - Gap

	            (*    Gap tail TO head function calculates the distance (Gap) between two parcels.
	                  The function increases the Counter WHILE the photo eye is clear.
	                  Everytime a parcel trigger the photo eye, gap value is save AND the counter is reset.  *)
	            IF NOT #sx_ReverseDirection
	            THEN
	                REGION 7.3.1 - Forward

	                    IF #ix_PECEoS       // Count displacement when the PE do not detects the product
	                    THEN

	                        IF #sdi_AuxGapTailtoHeadCounterFwd < #ci_OverflowLimit        // Prevent integer variable overflow
	                        THEN
	                            IF #iqUDT_HandShake.RTR THEN
	                                #sdi_AuxGapTailtoHeadCounterFwd += #iqUDT_ConveyorInterface.Displacement;    // Calculate the gap
	                            END_IF;

	                        END_IF;

	                    END_IF;

	                END_REGION
	            ELSE
	                REGION 7.3.2 - Reverse

	                    IF #ix_PECBoS       // Count displacement when the PE do not detects the product
	                    THEN

	                        IF #sdi_AuxGapTailtoHeadCounterRvs < #ci_OverflowLimit        // Prevent integer variable overflow
	                        THEN

	                            #sdi_AuxGapTailtoHeadCounterRvs -= #iqUDT_ConveyorInterface.Displacement;    // Calculate the gap

	                        END_IF;
	                    END_IF;

	                END_REGION
	            END_IF;
	        END_REGION

	        REGION 7.4 - Head to head

	            // The functionality head to head is used to calculate the distance between one head's parcel and the head's parcel behind.
	            // To do it, everytime the PEC is triggered, the function save the distance calculated and reset the counter to start
	            // counting again, over and over again.
	            IF NOT #sx_ReverseDirection
	            THEN
	                REGION 7.4.1 - Forward

	                    IF #sdi_AuxGapHeadToHeadCounterFwd < #ci_OverflowLimit        // Prevent integer variable overflow
	                    THEN

	                        #sdi_AuxGapHeadToHeadCounterFwd += #iqUDT_ConveyorInterface.Displacement;   // measure the distance between two products

	                    END_IF;

	                END_REGION
	            ELSE
	                REGION 7.4.2 - Reverse

	                    IF #sdi_AuxGapHeadToHeadCounterRvs < #ci_OverflowLimit        // Prevent integer variable overflow
	                    THEN

	                        #sdi_AuxGapHeadToHeadCounterRvs -= #iqUDT_ConveyorInterface.Displacement;   // measure the distance between two products

	                    END_IF;

	                END_REGION
	            END_IF;
	        END_REGION

	        REGION 7.5 - Check gaps between products

